C07227=1047.731,387.516,-124.764,173.908,41.828,158.146
C07228=1047.739,387.762,-124.805,173.915,41.833,158.148
C07229=1047.748,388.008,-124.847,173.922,41.839,158.150
C07230=1047.757,388.255,-124.889,173.929,41.845,158.152
C07231=1047.766,388.500,-124.931,173.936,41.851,158.154
C07232=1047.773,388.746,-124.973,173.943,41.857,158.155
C07233=1047.782,388.993,-125.015,173.951,41.863,158.157
C07234=1047.791,389.239,-125.057,173.957,41.869,158.159
C07235=1047.799,389.482,-125.099,173.964,41.874,158.161
C07236=1047.807,389.726,-125.140,173.972,41.880,158.163
C07237=1047.816,389.969,-125.182,173.979,41.887,158.165
C07238=1047.824,390.213,-125.224,173.985,41.893,158.167
C07239=1047.833,390.456,-125.266,173.992,41.898,158.169
C07240=1047.840,390.700,-125.307,174.000,41.904,158.171
C07241=1047.849,390.943,-125.350,174.007,41.910,158.173
C07242=1047.858,391.187,-125.392,174.014,41.917,158.175
C07243=1047.871,391.561,-125.456,174.025,41.926,158.178
C07244=1047.884,391.936,-125.521,174.036,41.935,158.181
C07245=1047.896,392.311,-125.586,174.047,41.944,158.184
C07246=1047.910,392.686,-125.651,174.058,41.954,158.187
C07247=1047.918,392.932,-125.693,174.065,41.960,158.189
C07248=1047.927,393.178,-125.736,174.073,41.966,158.191
C07249=1047.936,393.424,-125.779,174.080,41.972,158.193
C07250=1047.944,393.670,-125.822,174.088,41.979,158.195
C07251=1047.953,393.916,-125.865,174.095,41.985,158.197
C07252=1047.961,394.163,-125.907,174.103,41.991,158.199
C07253=1047.970,394.409,-125.950,174.110,41.997,158.201
C07254=1047.979,394.655,-125.993,174.118,42.004,158.203
C07255=1047.987,394.901,-126.036,174.125,42.010,158.205
C07256=1047.996,395.147,-126.079,174.133,42.017,158.207
C07257=1048.004,395.393,-126.122,174.140,42.023,158.209
C07258=1048.013,395.639,-126.165,174.148,42.029,158.212
C07259=1048.022,395.885,-126.207,174.155,42.035,158.214
C07260=1048.031,396.131,-126.251,174.163,42.042,158.216
C07261=1048.040,396.377,-126.294,174.170,42.048,158.218
C07262=1048.048,396.623,-126.337,174.178,42.055,158.220
C07263=1048.057,396.869,-126.380,174.185,42.062,158.222
C07264=1048.066,397.114,-126.424,174.193,42.068,158.224
C07265=1048.074,397.360,-126.467,174.200,42.074,158.226
C07266=1048.083,397.607,-126.510,174.209,42.081,158.228
C07267=1048.092,397.853,-126.554,174.217,42.087,158.231
C07268=1048.101,398.099,-126.597,174.224,42.094,158.233
C07269=1048.109,398.344,-126.641,174.232,42.101,158.235
C07270=1048.119,398.591,-126.684,174.240,42.107,158.237
C07271=1048.127,398.836,-126.728,174.247,42.114,158.239
C07272=1048.136,399.082,-126.771,174.255,42.121,158.242
C07273=1048.145,399.328,-126.815,174.263,42.127,158.244
C07274=1048.154,399.574,-126.858,174.271,42.134,158.246
C07275=1048.162,399.821,-126.903,174.279,42.141,158.248
C07276=1048.171,400.066,-126.947,174.287,42.147,158.250
C07277=1048.180,400.312,-126.990,174.294,42.154,158.253
C07278=1048.189,400.559,-127.034,174.303,42.161,158.255
C07279=1048.198,400.804,-127.078,174.311,42.167,158.257
C07280=1048.207,401.050,-127.122,174.318,42.174,158.259
C07281=1048.216,401.296,-127.165,174.326,42.181,158.262
C07282=1048.225,401.542,-127.209,174.335,42.188,158.264
C07283=1048.234,401.788,-127.253,174.343,42.195,158.266
C07284=1048.243,402.034,-127.297,174.350,42.201,158.268
C07285=1048.252,402.280,-127.341,174.359,42.208,158.271
C07286=1048.261,402.526,-127.385,174.367,42.215,158.273
C07287=1048.270,402.772,-127.429,174.375,42.222,158.275
C07288=1048.279,403.018,-127.474,174.384,42.229,158.278
C07289=1048.288,403.264,-127.518,174.391,42.236,158.280
C07290=1048.298,403.509,-127.563,174.399,42.243,158.282
C07291=1048.311,403.897,-127.633,174.413,42.254,158.286
C07292=1048.326,404.285,-127.702,174.425,42.265,158.290
C07293=1048.340,404.673,-127.773,174.439,42.276,158.294
C07294=1048.354,405.061,-127.843,174.452,42.288,158.297
C07295=1048.363,405.308,-127.887,174.461,42.295,158.300
C07296=1048.372,405.553,-127.932,174.468,42.302,158.302
C07297=1048.381,405.799,-127.978,174.478,42.309,158.305
C07298=1048.390,406.044,-128.021,174.485,42.316,158.307
C07299=1048.399,406.290,-128.067,174.495,42.324,158.310
C07300=1048.409,406.536,-128.111,174.502,42.331,158.312
C07301=1048.417,406.782,-128.156,174.511,42.338,158.314
C07302=1048.427,407.028,-128.201,174.519,42.345,158.317
C07303=1048.436,407.274,-128.246,174.528,42.353,158.319
C07304=1048.446,407.520,-128.291,174.537,42.360,158.322
C07305=1048.455,407.765,-128.336,174.545,42.367,158.324
C07306=1048.464,408.011,-128.381,174.555,42.374,158.327
C07307=1048.473,408.257,-128.426,174.563,42.382,158.329
C07308=1048.483,408.502,-128.471,174.572,42.389,158.332
C07309=1048.492,408.748,-128.517,174.580,42.397,158.334
C07310=1048.502,408.994,-128.561,174.589,42.404,158.337
C07311=1048.511,409.239,-128.607,174.598,42.412,158.339
C07312=1048.520,409.485,-128.652,174.606,42.419,158.342
C07313=1048.529,409.731,-128.697,174.615,42.427,158.344
C07314=1048.539,409.976,-128.742,174.625,42.434,158.347
C07315=1048.548,410.222,-128.787,174.633,42.442,158.350
C07316=1048.557,410.468,-128.833,174.642,42.449,158.352
C07317=1048.567,410.714,-128.878,174.651,42.456,158.355
C07318=1048.577,410.959,-128.924,174.660,42.464,158.357
C07319=1048.586,411.205,-128.969,174.669,42.472,158.360
C07320=1048.595,411.451,-129.014,174.678,42.479,158.362
C07321=1048.606,411.696,-129.060,174.687,42.487,158.365
C07322=1048.615,411.942,-129.106,174.696,42.495,158.368
C07323=1048.624,412.187,-129.152,174.705,42.502,158.370
C07324=1048.635,412.433,-129.197,174.715,42.510,158.373
C07325=1048.643,412.679,-129.242,174.724,42.518,158.376
C07326=1048.653,412.925,-129.288,174.732,42.526,158.378
C07327=1048.663,413.170,-129.335,174.742,42.534,158.381
C07328=1048.672,413.416,-129.380,174.751,42.541,158.384
C07329=1048.682,413.662,-129.426,174.761,42.549,158.387
C07330=1048.692,413.907,-129.472,174.770,42.557,158.389
C07331=1048.701,414.152,-129.519,174.779,42.565,158.392
C07332=1048.711,414.398,-129.565,174.789,42.573,158.395
C07333=1048.720,414.643,-129.611,174.798,42.581,158.397
C07334=1048.730,414.889,-129.658,174.807,42.589,158.400
C07335=1048.739,415.134,-129.704,174.817,42.597,158.403
C07336=1048.749,415.380,-129.750,174.826,42.604,158.406
C07337=1048.758,415.626,-129.796,174.836,42.613,158.409
C07338=1048.769,415.871,-129.842,174.845,42.621,158.411
C07339=1048.778,416.116,-129.889,174.855,42.629,158.414
C07340=1048.788,416.362,-129.935,174.864,42.637,158.417
C07341=1048.797,416.607,-129.981,174.874,42.645,158.420
C07342=1048.808,416.853,-130.028,174.883,42.653,158.423
C07343=1048.817,417.099,-130.075,174.893,42.662,158.425
C07344=1048.827,417.344,-130.121,174.903,42.669,158.428
C07345=1048.837,417.589,-130.168,174.913,42.678,158.431
C07346=1048.847,417.835,-130.215,174.923,42.686,158.434
C07347=1048.862,418.230,-130.290,174.939,42.699,158.439
C07348=1048.879,418.625,-130.365,174.954,42.712,158.443
C07349=1048.895,419.020,-130.441,174.970,42.726,158.448
C07350=1048.911,419.415,-130.517,174.986,42.740,158.453
C07351=1048.921,419.660,-130.563,174.996,42.748,158.456
C07352=1048.930,419.906,-130.611,175.007,42.756,158.459
C07353=1048.940,420.152,-130.658,175.017,42.765,158.462
C07354=1048.950,420.397,-130.705,175.026,42.774,158.465
C07355=1048.960,420.642,-130.752,175.037,42.782,158.468
C07356=1048.971,420.887,-130.799,175.047,42.791,158.471
C07357=1048.980,421.133,-130.847,175.058,42.799,158.474
C07358=1048.990,421.378,-130.894,175.068,42.808,158.477
C07359=1049.001,421.623,-130.942,175.078,42.816,158.480
C07360=1049.011,421.868,-130.990,175.088,42.825,158.483
C07361=1049.020,422.114,-131.037,175.098,42.834,158.486
C07362=1049.031,422.359,-131.085,175.109,42.842,158.489
C07363=1049.041,422.604,-131.132,175.119,42.851,158.492
C07364=1049.051,422.849,-131.180,175.130,42.860,158.495
C07365=1049.061,423.094,-131.227,175.141,42.868,158.499
C07366=1049.071,423.339,-131.275,175.151,42.878,158.502
C07367=1049.082,423.585,-131.323,175.162,42.886,158.505
C07368=1049.093,423.830,-131.371,175.172,42.895,158.508
C07369=1049.103,424.075,-131.418,175.183,42.904,158.511
C07370=1049.112,424.320,-131.467,175.194,42.913,158.514
C07371=1049.123,424.566,-131.514,175.204,42.922,158.518
C07372=1049.134,424.811,-131.562,175.215,42.931,158.521
C07373=1049.144,425.056,-131.611,175.226,42.939,158.524
C07374=1049.154,425.302,-131.658,175.236,42.949,158.527
C07375=1049.165,425.546,-131.706,175.247,42.957,158.530
C07376=1049.175,425.792,-131.755,175.259,42.966,158.534
C07377=1049.186,426.037,-131.803,175.270,42.976,158.537
C07378=1049.195,426.282,-131.852,175.280,42.985,158.540
C07379=1049.207,426.527,-131.900,175.291,42.994,158.544
C07380=1049.216,426.772,-131.948,175.303,43.003,158.547
C07381=1049.227,427.017,-131.997,175.314,43.012,158.550
C07382=1049.237,427.262,-132.046,175.325,43.021,158.554
C07383=1049.249,427.507,-132.094,175.336,43.031,158.557
C07384=1049.258,427.752,-132.143,175.348,43.040,158.560
C07385=1049.269,427.997,-132.191,175.359,43.049,158.564
C07386=1049.279,428.242,-132.240,175.369,43.059,158.567
C07387=1049.291,428.487,-132.289,175.381,43.068,158.571
C07388=1049.301,428.732,-132.338,175.392,43.078,158.574
C07389=1049.311,428.977,-132.387,175.403,43.087,158.577
C07390=1049.322,429.222,-132.436,175.416,43.096,158.581
C07391=1049.332,429.467,-132.484,175.427,43.106,158.584
C07392=1049.344,429.712,-132.533,175.439,43.116,158.588
C07393=1049.354,429.957,-132.583,175.450,43.125,158.591
C07394=1049.365,430.202,-132.633,175.462,43.135,158.595
C07395=1049.375,430.447,-132.681,175.473,43.144,158.599
C07396=1049.385,430.692,-132.731,175.485,43.154,158.602
C07397=1049.397,430.937,-132.780,175.496,43.163,158.606
C07398=1049.407,431.182,-132.829,175.508,43.173,158.609
C07399=1049.417,431.426,-132.879,175.521,43.183,158.613
C07400=1049.428,431.671,-132.928,175.532,43.193,158.616
C07401=1049.440,431.915,-132.978,175.544,43.203,158.620
C07402=1049.451,432.160,-133.027,175.557,43.212,158.624
C07403=1049.459,432.370,-133.070,175.567,43.221,158.627
C07404=1049.469,432.579,-133.112,175.577,43.229,158.630
C07405=1049.478,432.788,-133.155,175.587,43.237,158.633
C07406=1049.487,432.997,-133.197,175.598,43.246,158.636
C07407=1049.498,433.207,-133.240,175.608,43.254,158.639
C07408=1049.507,433.416,-133.283,175.618,43.263,158.642
C07409=1049.516,433.625,-133.325,175.629,43.271,158.646
C07410=1049.525,433.834,-133.368,175.639,43.280,158.649
C07411=1049.536,434.079,-133.417,175.651,43.290,158.653
C07412=1049.547,434.323,-133.467,175.664,43.300,158.656
C07413=1049.559,434.569,-133.518,175.676,43.310,158.660
C07414=1049.570,434.813,-133.568,175.689,43.320,158.664
C07415=1049.581,435.058,-133.618,175.702,43.330,158.668
C07416=1049.592,435.302,-133.668,175.714,43.341,158.672
C07417=1049.604,435.547,-133.718,175.726,43.351,158.675
C07418=1049.615,435.792,-133.769,175.739,43.361,158.679
C07419=1049.626,436.036,-133.819,175.752,43.371,158.683
C07420=1049.637,436.281,-133.870,175.764,43.381,158.687
C07421=1049.648,436.526,-133.920,175.778,43.391,158.691
C07422=1049.659,436.770,-133.970,175.790,43.402,158.695
C07423=1049.671,437.015,-134.021,175.803,43.412,158.699
C07424=1049.682,437.259,-134.072,175.816,43.423,158.703
C07425=1049.694,437.504,-134.123,175.829,43.433,158.707
C07426=1049.705,437.749,-134.173,175.841,43.444,158.711
C07427=1049.717,437.993,-134.224,175.855,43.455,158.715
C07428=1049.728,438.238,-134.275,175.868,43.465,158.719
C07429=1049.740,438.482,-134.326,175.881,43.476,158.723
C07430=1049.750,438.727,-134.376,175.894,43.486,158.727
C07431=1049.762,438.971,-134.428,175.908,43.497,158.731
C07432=1049.774,439.216,-134.480,175.921,43.508,158.735
C07433=1049.785,439.460,-134.531,175.935,43.518,158.739
C07434=1049.797,439.704,-134.582,175.948,43.529,158.743
C07435=1049.808,439.949,-134.633,175.961,43.540,158.747
C07436=1049.820,440.193,-134.684,175.975,43.551,158.751
C07437=1049.831,440.438,-134.736,175.988,43.562,158.756
C07438=1049.843,440.682,-134.788,176.002,43.573,158.760
C07439=1049.855,440.926,-134.840,176.016,43.583,158.764
C07440=1049.866,441.170,-134.891,176.030,43.594,158.768
C07441=1049.878,441.415,-134.942,176.043,43.605,158.772
C07442=1049.890,441.659,-134.993,176.057,43.616,158.777
C07443=1049.901,441.903,-135.046,176.072,43.627,158.781
C07444=1049.913,442.148,-135.098,176.085,43.639,158.785
C07445=1049.925,442.392,-135.150,176.099,43.650,158.790
C07446=1049.936,442.637,-135.202,176.114,43.661,158.794
C07447=1049.949,442.880,-135.254,176.128,43.672,158.798
C07448=1049.961,443.124,-135.306,176.141,43.683,158.803
C07449=1049.973,443.369,-135.357,176.156,43.695,158.807
C07450=1049.984,443.613,-135.410,176.170,43.706,158.812
C07451=1049.996,443.857,-135.462,176.185,43.717,158.816
C07452=1050.009,444.101,-135.514,176.199,43.729,158.821
C07453=1050.020,444.345,-135.567,176.214,43.740,158.825
C07454=1050.033,444.590,-135.619,176.229,43.752,158.830
C07455=1050.045,444.834,-135.672,176.243,43.763,158.834
C07456=1050.056,445.078,-135.724,176.258,43.775,158.839
C07457=1050.069,445.322,-135.777,176.273,43.786,158.843
C07458=1050.081,445.566,-135.829,176.287,43.798,158.848
C07459=1050.093,445.809,-135.881,176.302,43.809,158.852
C07460=1050.106,446.052,-135.934,176.317,43.821,158.857
C07461=1050.119,446.296,-135.986,176.332,43.832,158.862
C07462=1050.132,446.540,-136.038,176.347,43.843,158.866
C07463=1050.148,446.805,-136.093,176.364,43.856,158.871
C07464=1050.165,447.073,-136.149,176.380,43.868,158.876
C07465=1050.182,447.340,-136.203,176.396,43.879,158.881
C07466=1050.201,447.608,-136.257,176.414,43.891,158.886
C07467=1050.219,447.852,-136.306,176.430,43.901,158.890
C07468=1050.237,448.096,-136.353,176.444,43.912,158.894
C07469=1050.255,448.341,-136.401,176.460,43.922,158.899
C07470=1050.275,448.586,-136.448,176.476,43.932,158.903
C07471=1050.296,448.830,-136.495,176.492,43.942,158.907
C07472=1050.317,449.075,-136.541,176.508,43.951,158.911
C07473=1050.338,449.321,-136.586,176.523,43.961,158.916
C07474=1050.361,449.566,-136.631,176.540,43.971,158.920
C07475=1050.384,449.811,-136.675,176.556,43.980,158.924
C07476=1050.408,450.056,-136.719,176.572,43.989,158.928
C07477=1050.432,450.302,-136.762,176.588,43.998,158.932
C07478=1050.458,450.546,-136.805,176.605,44.007,158.936
C07479=1050.144,450.574,-137.105,176.604,44.099,158.963
C07480=1050.118,450.329,-137.062,176.588,44.090,158.959
C07481=1050.094,450.083,-137.019,176.572,44.081,158.955
C07482=1050.070,449.838,-136.975,176.556,44.073,158.951
C07483=1050.046,449.593,-136.931,176.539,44.064,158.947
C07484=1050.024,449.348,-136.887,176.523,44.054,158.942
C07485=1050.002,449.103,-136.841,176.507,44.044,158.938
C07486=1049.981,448.858,-136.795,176.492,44.034,158.934
C07487=1049.960,448.613,-136.749,176.475,44.025,158.930
C07488=1049.941,448.368,-136.702,176.460,44.015,158.925
C07489=1049.921,448.124,-136.654,176.444,44.005,158.921
C07490=1049.903,447.880,-136.607,176.428,43.995,158.917
C07491=1049.886,447.636,-136.558,176.412,43.985,158.912
C07492=1049.868,447.386,-136.507,176.397,43.973,158.908
C07493=1049.851,447.137,-136.457,176.381,43.963,158.903
C07494=1049.836,446.888,-136.406,176.365,43.952,158.899
C07495=1049.821,446.639,-136.354,176.350,43.940,158.894
C07496=1049.806,446.395,-136.303,176.335,43.929,158.890
C07497=1049.792,446.151,-136.251,176.320,43.918,158.885
C07498=1049.779,445.908,-136.199,176.305,43.907,158.881
C07499=1049.767,445.666,-136.147,176.290,43.895,158.876
C07500=1049.755,445.422,-136.094,176.275,43.884,158.871
C07501=1049.743,445.177,-136.041,176.260,43.872,158.867
C07502=1049.730,444.933,-135.989,176.246,43.861,158.862
C07503=1049.719,444.690,-135.936,176.231,43.850,158.858
C07504=1049.706,444.446,-135.884,176.216,43.838,158.853
C07505=1049.694,444.201,-135.831,176.202,43.826,158.849
C07506=1049.682,443.957,-135.779,176.187,43.816,158.844
C07507=1049.670,443.713,-135.726,176.173,43.804,158.840
C07508=1049.658,443.469,-135.675,176.158,43.793,158.835
C07509=1049.647,443.224,-135.622,176.144,43.782,158.831
C07510=1049.635,442.980,-135.570,176.129,43.770,158.826
C07511=1049.622,442.737,-135.518,176.115,43.759,158.822
C07512=1049.611,442.492,-135.466,176.101,43.748,158.818
C07513=1049.599,442.248,-135.414,176.087,43.737,158.813
C07514=1049.587,442.003,-135.363,176.072,43.726,158.809
C07515=1049.575,441.759,-135.310,176.059,43.715,158.805
C07516=1049.564,441.515,-135.258,176.045,43.704,158.800
C07517=1049.552,441.270,-135.207,176.030,43.693,158.796
C07518=1049.540,441.026,-135.155,176.017,43.682,158.792
C07519=1049.528,440.782,-135.104,176.003,43.672,158.788
C07520=1049.516,440.537,-135.052,175.989,43.660,158.783
C07521=1049.504,440.293,-135.001,175.976,43.650,158.779
C07522=1049.494,440.049,-134.949,175.962,43.639,158.775
C07523=1049.482,439.804,-134.898,175.948,43.628,158.771
C07524=1049.470,439.560,-134.846,175.935,43.618,158.767
C07525=1049.458,439.316,-134.795,175.921,43.607,158.763
C07526=1049.447,439.071,-134.744,175.908,43.596,158.759
C07527=1049.435,438.826,-134.693,175.894,43.585,158.754
C07528=1049.424,438.582,-134.642,175.881,43.575,158.750
C07529=1049.413,438.337,-134.590,175.868,43.564,158.746
C07530=1049.401,438.092,-134.539,175.855,43.554,158.742
C07531=1049.390,437.849,-134.488,175.841,43.543,158.738
C07532=1049.378,437.603,-134.438,175.829,43.533,158.734
C07533=1049.367,437.360,-134.387,175.816,43.522,158.730
C07534=1049.355,437.114,-134.336,175.803,43.512,158.726
C07535=1049.344,436.870,-134.286,175.789,43.502,158.722
C07536=1049.333,436.626,-134.235,175.776,43.492,158.718
C07537=1049.322,436.381,-134.184,175.764,43.481,158.715
C07538=1049.311,436.137,-134.134,175.751,43.471,158.711
C07539=1049.299,435.892,-134.083,175.738,43.460,158.707
C07540=1049.287,435.647,-134.033,175.725,43.451,158.703
C07541=1049.276,435.403,-133.983,175.713,43.440,158.699
C07542=1049.265,435.158,-133.932,175.700,43.430,158.695
C07543=1049.254,434.913,-133.883,175.687,43.420,158.691
C07544=1049.243,434.668,-133.832,175.675,43.410,158.688
C07545=1049.231,434.424,-133.782,175.662,43.400,158.684
C07546=1049.220,434.180,-133.732,175.650,43.390,158.680
C07547=1049.209,433.934,-133.682,175.637,43.380,158.676
C07548=1049.200,433.724,-133.639,175.627,43.372,158.673
C07549=1049.190,433.514,-133.596,175.616,43.363,158.670
C07550=1049.180,433.304,-133.554,175.606,43.355,158.667
C07551=1049.171,433.094,-133.511,175.596,43.346,158.663
C07552=1049.161,432.884,-133.468,175.585,43.338,158.660
C07553=1049.152,432.673,-133.425,175.574,43.329,158.657
C07554=1049.143,432.463,-133.382,175.563,43.321,158.654
C07555=1049.134,432.253,-133.340,175.553,43.313,158.651
C07556=1049.123,432.008,-133.290,175.542,43.302,158.647
C07557=1049.112,431.764,-133.241,175.530,43.293,158.644
C07558=1049.101,431.519,-133.191,175.517,43.283,158.640
C07559=1049.090,431.274,-133.141,175.506,43.273,158.636
C07560=1049.080,431.029,-133.092,175.494,43.264,158.633
C07561=1049.068,430.784,-133.043,175.482,43.254,158.629
C07562=1049.058,430.539,-132.993,175.470,43.244,158.626
C07563=1049.048,430.294,-132.944,175.458,43.235,158.622
C07564=1049.037,430.049,-132.894,175.447,43.225,158.618
C07565=1049.026,429.804,-132.846,175.435,43.216,158.615
C07566=1049.015,429.559,-132.796,175.424,43.207,158.612
C07567=1049.005,429.315,-132.747,175.412,43.197,158.608
C07568=1048.994,429.070,-132.698,175.401,43.187,158.605
C07569=1048.983,428.824,-132.649,175.389,43.178,158.601
C07570=1048.973,428.578,-132.600,175.377,43.169,158.598
C07571=1048.962,428.334,-132.552,175.366,43.160,158.594
C07572=1048.952,428.089,-132.503,175.354,43.150,158.591
C07573=1048.941,427.845,-132.454,175.343,43.141,158.587
C07574=1048.931,427.599,-132.405,175.332,43.132,158.584
C07575=1048.920,427.354,-132.357,175.321,43.123,158.581
C07576=1048.909,427.109,-132.308,175.310,43.113,158.577
C07577=1048.898,426.864,-132.259,175.298,43.104,158.574
C07578=1048.889,426.619,-132.211,175.287,43.095,158.571
C07579=1048.878,426.374,-132.163,175.276,43.086,158.567
C07580=1048.868,426.129,-132.114,175.265,43.077,158.564
C07581=1048.857,425.884,-132.066,175.254,43.068,158.561
C07582=1048.847,425.638,-132.017,175.243,43.059,158.557
C07583=1048.836,425.394,-131.969,175.232,43.050,158.554
C07584=1048.826,425.149,-131.921,175.221,43.041,158.551
C07585=1048.816,424.903,-131.872,175.210,43.032,158.548
C07586=1048.805,424.658,-131.825,175.200,43.023,158.545
C07587=1048.794,424.413,-131.777,175.189,43.014,158.541
C07588=1048.785,424.168,-131.728,175.178,43.005,158.538
C07589=1048.774,423.922,-131.681,175.168,42.997,158.535
C07590=1048.764,423.678,-131.633,175.157,42.988,158.532
C07591=1048.753,423.432,-131.586,175.146,42.979,158.529
C07592=1048.743,423.187,-131.537,175.135,42.970,158.525
C07593=1048.733,422.942,-131.490,175.124,42.961,158.522
C07594=1048.723,422.697,-131.442,175.114,42.953,158.519
C07595=1048.712,422.452,-131.395,175.104,42.944,158.516
C07596=1048.703,422.206,-131.347,175.093,42.936,158.513
C07597=1048.693,421.961,-131.300,175.083,42.927,158.510
C07598=1048.682,421.716,-131.252,175.072,42.918,158.507
C07599=1048.671,421.470,-131.204,175.062,42.910,158.504
C07600=1048.661,421.225,-131.157,175.052,42.901,158.501
C07601=1048.652,420.980,-131.110,175.041,42.893,158.498
C07602=1048.642,420.735,-131.062,175.031,42.884,158.495
C07603=1048.632,420.489,-131.015,175.020,42.876,158.491
C07604=1048.622,420.244,-130.968,175.011,42.867,158.489
C07605=1048.612,419.999,-130.921,175.001,42.859,158.486
C07606=1048.602,419.753,-130.873,174.990,42.850,158.482
C07607=1048.592,419.508,-130.826,174.980,42.842,158.480
C07608=1048.576,419.111,-130.750,174.964,42.828,158.475
C07609=1048.560,418.714,-130.674,174.947,42.815,158.470
C07610=1048.544,418.317,-130.598,174.931,42.801,158.465
C07611=1048.528,417.920,-130.523,174.915,42.788,158.461
C07612=1048.517,417.674,-130.476,174.906,42.780,158.458
C07613=1048.508,417.429,-130.429,174.896,42.772,158.455
C07614=1048.498,417.183,-130.383,174.886,42.764,158.452
C07615=1048.488,416.938,-130.336,174.876,42.756,158.449
C07616=1048.478,416.692,-130.289,174.866,42.748,158.446
C07617=1048.468,416.446,-130.243,174.857,42.740,158.443
C07618=1048.459,416.202,-130.196,174.847,42.731,158.441
C07619=1048.449,415.956,-130.149,174.838,42.724,158.438
C07620=1048.440,415.711,-130.103,174.828,42.715,158.435
C07621=1048.430,415.465,-130.057,174.819,42.707,158.432
C07622=1048.419,415.219,-130.011,174.809,42.700,158.429
C07623=1048.410,414.974,-129.965,174.800,42.692,158.427
C07624=1048.400,414.728,-129.918,174.790,42.684,158.424
C07625=1048.391,414.483,-129.872,174.781,42.676,158.421
C07626=1048.381,414.238,-129.826,174.771,42.668,158.418
C07627=1048.371,413.992,-129.779,174.762,42.660,158.416
C07628=1048.362,413.746,-129.733,174.753,42.652,158.413
C07629=1048.352,413.501,-129.687,174.743,42.645,158.410
C07630=1048.343,413.255,-129.641,174.734,42.637,158.407
C07631=1048.333,413.010,-129.596,174.724,42.629,158.405
C07632=1048.323,412.764,-129.549,174.715,42.621,158.402
C07633=1048.314,412.518,-129.504,174.706,42.614,158.399
C07634=1048.304,412.272,-129.457,174.696,42.606,158.397
C07635=1048.295,412.027,-129.413,174.687,42.598,158.394
C07636=1048.285,411.781,-129.366,174.679,42.590,158.391
C07637=1048.275,411.535,-129.321,174.670,42.583,158.389
C07638=1048.266,411.289,-129.276,174.660,42.575,158.386
C07639=1048.257,411.044,-129.230,174.651,42.568,158.384
C07640=1048.247,410.799,-129.185,174.642,42.560,158.381
C07641=1048.238,410.552,-129.139,174.634,42.553,158.378
C07642=1048.228,410.307,-129.094,174.625,42.545,158.376
C07643=1048.219,410.061,-129.048,174.615,42.538,158.373
C07644=1048.209,409.816,-129.003,174.606,42.530,158.371
C07645=1048.200,409.570,-128.958,174.598,42.523,158.368
C07646=1048.190,409.325,-128.913,174.589,42.515,158.365
C07647=1048.181,409.078,-128.867,174.580,42.508,158.363
C07648=1048.171,408.833,-128.822,174.570,42.500,158.360
C07649=1048.162,408.587,-128.777,174.562,42.493,158.358
C07650=1048.152,408.341,-128.732,174.553,42.486,158.355
C07651=1048.143,408.095,-128.687,174.545,42.479,158.353
C07652=1048.134,407.850,-128.641,174.536,42.471,158.350
C07653=1048.125,407.604,-128.597,174.527,42.464,158.348
C07654=1048.116,407.358,-128.551,174.519,42.457,158.345
C07655=1048.106,407.112,-128.507,174.510,42.449,158.343
C07656=1048.097,406.866,-128.462,174.502,42.442,158.341
C07657=1048.088,406.622,-128.417,174.493,42.435,158.338
C07658=1048.079,406.376,-128.372,174.484,42.428,158.336
C07659=1048.070,406.130,-128.328,174.476,42.420,158.333
C07660=1048.061,405.884,-128.282,174.467,42.414,158.331
C07661=1048.051,405.638,-128.238,174.459,42.407,158.328
C07662=1048.042,405.392,-128.193,174.450,42.399,158.326
C07663=1048.034,405.146,-128.149,174.442,42.392,158.323
C07664=1048.019,404.757,-128.078,174.428,42.381,158.320
C07665=1048.004,404.366,-128.007,174.415,42.370,158.316
C07666=1047.990,403.976,-127.936,174.402,42.359,158.312
C07667=1047.976,403.586,-127.866,174.389,42.348,158.308
C07668=1047.967,403.341,-127.822,174.380,42.341,158.306
C07669=1047.958,403.095,-127.777,174.373,42.334,158.304
C07670=1047.948,402.849,-127.733,174.364,42.327,158.301
C07671=1047.940,402.603,-127.689,174.356,42.320,158.299
C07672=1047.931,402.357,-127.645,174.348,42.313,158.297
C07673=1047.921,402.111,-127.600,174.339,42.306,158.295
C07674=1047.913,401.865,-127.557,174.331,42.299,158.292
C07675=1047.903,401.619,-127.513,174.324,42.293,158.290
C07676=1047.894,401.374,-127.469,174.315,42.286,158.288
C07677=1047.886,401.127,-127.424,174.307,42.279,158.285
C07678=1047.877,400.882,-127.380,174.299,42.272,158.283
C07679=1047.868,400.635,-127.337,174.292,42.266,158.281
C07680=1047.859,400.389,-127.293,174.283,42.259,158.279
C07681=1047.850,400.143,-127.249,174.275,42.252,158.276
C07682=1047.841,399.898,-127.205,174.267,42.246,158.274
C07683=1047.832,399.651,-127.162,174.260,42.239,158.272
C07684=1047.823,399.406,-127.118,174.251,42.232,158.270
C07685=1047.814,399.160,-127.075,174.243,42.226,158.268
C07686=1047.805,398.914,-127.031,174.236,42.219,158.265
C07687=1047.796,398.668,-126.987,174.228,42.213,158.263
C07688=1047.788,398.422,-126.944,174.220,42.206,158.261
C07689=1047.778,398.176,-126.900,174.213,42.199,158.259
C07690=1047.770,397.930,-126.857,174.204,42.193,158.257
C07691=1047.761,397.684,-126.814,174.197,42.187,158.254
C07692=1047.752,397.438,-126.770,174.189,42.180,158.252
C07693=1047.743,397.192,-126.727,174.181,42.173,158.250
C07694=1047.735,396.946,-126.683,174.174,42.167,158.248
C07695=1047.726,396.700,-126.640,174.166,42.160,158.246
C07696=1047.718,396.454,-126.597,174.159,42.154,158.244
C07697=1047.708,396.207,-126.554,174.151,42.148,158.242
C07698=1047.700,395.962,-126.510,174.143,42.141,158.239
C07699=1047.691,395.716,-126.467,174.135,42.135,158.237
C07700=1047.683,395.470,-126.424,174.127,42.129,158.235
C07701=1047.673,395.224,-126.382,174.120,42.122,158.233
C07702=1047.665,394.978,-126.339,174.112,42.116,158.231
C07703=1047.656,394.732,-126.296,174.105,42.110,158.229
C07704=1047.647,394.485,-126.252,174.097,42.104,158.227
C07705=1047.639,394.239,-126.209,174.090,42.097,158.225
C07706=1047.630,393.993,-126.167,174.082,42.091,158.223
C07707=1047.621,393.747,-126.124,174.075,42.085,158.221
C07708=1047.613,393.501,-126.081,174.067,42.078,158.219
C07709=1047.604,393.255,-126.038,174.060,42.072,158.217
C07710=1047.596,393.009,-125.995,174.052,42.066,158.215
C07711=1047.587,392.763,-125.953,174.045,42.060,158.213
C07712=1047.578,392.517,-125.910,174.039,42.054,158.211
C07713=1047.571,392.271,-125.868,174.031,42.047,158.209
C07714=1047.562,392.025,-125.825,174.024,42.041,158.207
C07715=1047.553,391.779,-125.782,174.016,42.035,158.205
C07716=1047.545,391.532,-125.740,174.009,42.029,158.203
C07717=1047.536,391.286,-125.697,174.001,42.023,158.201
C07718=1047.527,391.040,-125.655,173.994,42.017,158.199
C07719=1047.519,390.794,-125.612,173.987,42.011,158.197
C07720=1047.506,390.422,-125.549,173.976,42.002,158.194
C07721=1047.493,390.051,-125.485,173.966,41.993,158.191
C07722=1047.480,389.680,-125.422,173.954,41.984,158.188
C07723=1047.468,389.309,-125.358,173.944,41.975,158.185
C07724=1047.459,389.062,-125.316,173.936,41.970,158.183
C07725=1047.451,388.816,-125.273,173.930,41.963,158.181
C07726=1047.441,388.570,-125.231,173.923,41.957,158.179
C07727=1047.434,388.324,-125.189,173.916,41.952,158.177
C07728=1047.425,388.078,-125.147,173.908,41.946,158.175
C07729=1047.416,387.831,-125.106,173.901,41.940,158.174
C07730=1047.408,387.584,-125.063,173.895,41.935,158.172
C07731=1047.399,387.339,-125.022,173.888,41.928,158.170
C07732=1047.391,387.092,-124.980,173.880,41.923,158.168
C07733=1047.382,386.846,-124.938,173.873,41.917,158.166
C07734=1047.374,386.600,-124.897,173.867,41.911,158.164
C07735=1047.365,386.354,-124.855,173.860,41.906,158.162
C07736=1047.357,386.106,-124.813,173.853,41.900,158.160
C07737=1047.349,385.861,-124.772,173.845,41.894,158.159
C07738=1047.340,385.614,-124.730,173.839,41.888,158.157
C07739=1047.332,385.368,-124.688,173.832,41.883,158.155
C07740=1047.323,385.122,-124.647,173.825,41.877,158.153
C07741=1047.315,384.876,-124.606,173.819,41.872,158.151
C07742=1047.307,384.629,-124.564,173.811,41.866,158.149
C07743=1047.298,384.383,-124.522,173.805,41.860,158.148
C07744=1047.290,384.136,-124.481,173.798,41.855,158.146
C07745=1047.282,383.890,-124.439,173.791,41.849,158.144
C07746=1047.274,383.644,-124.398,173.785,41.844,158.142
C07747=1047.266,383.398,-124.357,173.778,41.838,158.140
C07748=1047.257,383.151,-124.315,173.771,41.832,158.139
C07749=1047.249,382.905,-124.274,173.764,41.827,158.137
C07750=1047.240,382.659,-124.232,173.757,41.821,158.135
C07751=1047.232,382.412,-124.192,173.751,41.816,158.133
C07752=1047.225,382.165,-124.150,173.744,41.810,158.132
C07753=1047.216,381.919,-124.109,173.738,41.805,158.130
C07754=1047.208,381.673,-124.068,173.731,41.799,158.128
C07755=1047.200,381.426,-124.026,173.725,41.794,158.126
C07756=1047.192,381.180,-123.985,173.718,41.789,158.125
C07757=1047.184,380.934,-123.945,173.712,41.783,158.123
C07758=1047.175,380.687,-123.904,173.705,41.778,158.121
C07759=1047.168,380.441,-123.862,173.699,41.772,158.119
C07760=1047.160,380.195,-123.821,173.692,41.766,158.118
C07761=1047.152,379.948,-123.780,173.686,41.761,158.116
C07762=1047.144,379.701,-123.739,173.679,41.756,158.114
C07763=1047.136,379.455,-123.698,173.673,41.751,158.112
C07764=1047.128,379.208,-123.657,173.666,41.745,158.111
C07765=1047.120,378.962,-123.617,173.660,41.740,158.109
C07766=1047.111,378.715,-123.576,173.653,41.735,158.107
C07767=1047.103,378.469,-123.535,173.647,41.730,158.106
C07768=1047.094,378.212,-123.492,173.640,41.724,158.104
C07769=1047.086,377.954,-123.450,173.634,41.718,158.102
C07770=1047.077,377.698,-123.408,173.626,41.713,158.100
C07771=1047.069,377.440,-123.366,173.620,41.708,158.099
C07772=1047.061,377.194,-123.325,173.614,41.703,158.097
C07773=1047.053,376.947,-123.285,173.608,41.697,158.096
C07774=1047.044,376.700,-123.244,173.601,41.692,158.094
C07775=1047.036,376.453,-123.204,173.595,41.687,158.092
C07776=1047.025,376.126,-123.151,173.586,41.680,158.090
C07777=1047.015,375.798,-123.097,173.578,41.673,158.088
C07778=1047.004,375.472,-123.043,173.569,41.667,158.086
C07779=1046.994,375.144,-122.989,173.562,41.659,158.083
C07780=1046.986,374.897,-122.950,173.555,41.654,158.082
C07781=1046.978,374.651,-122.909,173.549,41.649,158.080
C07782=1046.970,374.404,-122.869,173.543,41.645,158.079
C07783=1046.962,374.158,-122.829,173.536,41.640,158.077
C07784=1046.954,373.911,-122.789,173.530,41.634,158.076
C07785=1046.946,373.665,-122.748,173.524,41.629,158.074
C07786=1046.938,373.418,-122.708,173.518,41.624,158.072
C07787=1046.931,373.171,-122.668,173.512,41.620,158.071
C07788=1046.923,372.925,-122.628,173.506,41.614,158.069
C07789=1046.915,372.678,-122.588,173.500,41.609,158.068
C07790=1046.906,372.431,-122.548,173.493,41.604,158.066
C07791=1046.899,372.186,-122.508,173.487,41.599,158.064
C07792=1046.891,371.939,-122.468,173.482,41.594,158.063
C07793=1046.884,371.692,-122.428,173.476,41.589,158.061
C07794=1046.876,371.445,-122.388,173.470,41.584,158.060
C07795=1046.868,371.198,-122.348,173.463,41.579,158.058
C07796=1046.860,370.951,-122.308,173.457,41.575,158.057
C07797=1046.852,370.705,-122.269,173.452,41.570,158.055
C07798=1046.844,370.458,-122.229,173.446,41.565,158.054
C07799=1046.836,370.211,-122.190,173.439,41.560,158.052
C07800=1046.829,369.965,-122.150,173.433,41.555,158.051
C07801=1046.821,369.718,-122.110,173.428,41.551,158.049
C07802=1046.812,369.471,-122.071,173.422,41.546,158.048
C07803=1046.805,369.224,-122.031,173.416,41.541,158.046
C07804=1046.796,368.978,-121.992,173.409,41.536,158.045
C07805=1046.789,368.732,-121.952,173.404,41.532,158.043
C07806=1046.781,368.485,-121.913,173.398,41.527,158.042
C07807=1046.773,368.237,-121.874,173.392,41.522,158.040
C07808=1046.765,367.991,-121.834,173.386,41.517,158.039
C07809=1046.758,367.745,-121.795,173.381,41.512,158.037
C07810=1046.750,367.498,-121.755,173.375,41.508,158.036
C07811=1046.742,367.251,-121.716,173.369,41.503,158.034
C07812=1046.734,367.004,-121.676,173.363,41.499,158.033
C07813=1046.726,366.758,-121.637,173.357,41.494,158.031
C07814=1046.719,366.510,-121.598,173.351,41.489,158.030
C07815=1046.710,366.264,-121.559,173.346,41.484,158.028
C07816=1046.704,366.017,-121.520,173.340,41.479,158.027
C07817=1046.695,365.770,-121.481,173.334,41.475,158.025
C07818=1046.688,365.524,-121.441,173.328,41.470,158.024
C07819=1046.680,365.277,-121.403,173.323,41.466,158.023
C07820=1046.672,365.030,-121.363,173.317,41.461,158.021
C07821=1046.665,364.783,-121.324,173.312,41.457,158.020
C07822=1046.657,364.536,-121.285,173.306,41.452,158.018
C07823=1046.650,364.290,-121.246,173.300,41.447,158.017
C07824=1046.642,364.042,-121.207,173.295,41.443,158.015
C07825=1046.635,363.796,-121.168,173.289,41.438,158.014
C07826=1046.627,363.549,-121.129,173.283,41.433,158.013
C07827=1046.620,363.302,-121.090,173.278,41.429,158.011
C07828=1046.611,363.056,-121.051,173.272,41.424,158.010
C07829=1046.605,362.809,-121.012,173.267,41.420,158.008
C07830=1046.596,362.562,-120.973,173.261,41.415,158.007
C07831=1046.589,362.315,-120.935,173.255,41.411,158.006
C07832=1046.578,361.996,-120.885,173.248,41.405,158.004
C07833=1046.568,361.677,-120.835,173.240,41.399,158.002
C07834=1046.559,361.358,-120.785,173.233,41.393,158.000
C07835=1046.549,361.040,-120.735,173.226,41.388,157.998
C07836=1046.541,360.792,-120.696,173.221,41.384,157.997
C07837=1046.534,360.546,-120.658,173.215,41.379,157.996
C07838=1046.526,360.299,-120.620,173.210,41.375,157.994
C07839=1046.518,360.052,-120.581,173.204,41.370,157.993
C07840=1046.511,359.805,-120.543,173.199,41.366,157.992
C07841=1046.504,359.557,-120.504,173.194,41.362,157.990
C07842=1046.496,359.311,-120.466,173.188,41.357,157.989
C07843=1046.488,359.064,-120.428,173.183,41.353,157.988
C07844=1046.480,358.817,-120.389,173.177,41.348,157.986
C07845=1046.473,358.570,-120.351,173.172,41.344,157.985
C07846=1046.466,358.324,-120.312,173.166,41.340,157.984
C07847=1046.458,358.076,-120.274,173.161,41.336,157.982
C07848=1046.451,357.829,-120.236,173.155,41.331,157.981
C07849=1046.443,357.583,-120.198,173.151,41.327,157.980
C07850=1046.435,357.335,-120.160,173.145,41.323,157.978
C07851=1046.428,357.088,-120.122,173.140,41.319,157.977
C07852=1046.420,356.842,-120.083,173.134,41.314,157.976
C07853=1046.413,356.595,-120.046,173.129,41.310,157.974
C07854=1046.405,356.348,-120.007,173.123,41.306,157.973
C07855=1046.397,356.100,-119.970,173.118,41.302,157.972
C07856=1046.390,355.854,-119.931,173.113,41.297,157.971
C07857=1046.383,355.607,-119.894,173.108,41.293,157.969
C07858=1046.374,355.360,-119.855,173.102,41.289,157.968
C07859=1046.367,355.112,-119.818,173.097,41.285,157.967
C07860=1046.360,354.866,-119.779,173.092,41.281,157.966
C07861=1046.352,354.619,-119.742,173.086,41.277,157.964
C07862=1046.345,354.372,-119.704,173.082,41.272,157.963
C07863=1046.337,354.124,-119.666,173.076,41.268,157.962
C07864=1046.330,353.877,-119.628,173.071,41.264,157.960
C07865=1046.322,353.631,-119.590,173.065,41.260,157.959
C07866=1046.315,353.384,-119.553,173.061,41.256,157.958
C07867=1046.308,353.137,-119.515,173.055,41.252,157.957
C07868=1046.300,352.889,-119.477,173.050,41.247,157.955
C07869=1046.293,352.643,-119.439,173.045,41.243,157.954
C07870=1046.286,352.396,-119.402,173.040,41.240,157.953
C07871=1046.278,352.148,-119.364,173.035,41.235,157.952
C07872=1046.271,351.901,-119.326,173.029,41.231,157.950
C07873=1046.263,351.654,-119.289,173.024,41.227,157.949
C07874=1046.256,351.406,-119.251,173.020,41.223,157.948
C07875=1046.249,351.160,-119.213,173.014,41.219,157.947
C07876=1046.241,350.913,-119.176,173.009,41.215,157.945
C07877=1046.233,350.666,-119.139,173.004,41.211,157.944
C07878=1046.226,350.419,-119.101,172.999,41.207,157.943
C07879=1046.219,350.172,-119.063,172.994,41.203,157.942
C07880=1046.212,349.925,-119.026,172.989,41.199,157.941
C07881=1046.204,349.677,-118.988,172.984,41.195,157.939
C07882=1046.197,349.430,-118.952,172.979,41.191,157.938
C07883=1046.189,349.183,-118.915,172.973,41.187,157.937
C07884=1046.182,348.936,-118.877,172.969,41.183,157.936
C07885=1046.174,348.689,-118.840,172.963,41.179,157.935
C07886=1046.167,348.442,-118.803,172.958,41.176,157.933
C07887=1046.160,348.195,-118.765,172.954,41.171,157.932
C07888=1046.151,347.882,-118.718,172.947,41.167,157.931
C07889=1046.141,347.569,-118.671,172.941,41.161,157.929
C07890=1046.132,347.255,-118.625,172.935,41.157,157.928
C07891=1046.123,346.941,-118.578,172.928,41.151,157.926
C07892=1046.116,346.694,-118.540,172.924,41.148,157.925
C07893=1046.108,346.447,-118.503,172.919,41.144,157.924
C07894=1046.101,346.200,-118.467,172.914,41.140,157.923
C07895=1046.094,345.953,-118.429,172.909,41.136,157.922
C07896=1046.086,345.706,-118.393,172.904,41.133,157.920
C07897=1046.079,345.459,-118.355,172.899,41.128,157.919
C07898=1046.071,345.212,-118.319,172.894,41.125,157.918
C07899=1046.064,344.964,-118.282,172.890,41.121,157.917
C07900=1046.057,344.718,-118.245,172.884,41.117,157.916
C07901=1046.050,344.470,-118.208,172.879,41.113,157.915
C07902=1046.043,344.223,-118.171,172.875,41.110,157.913
C07903=1046.035,343.975,-118.135,172.870,41.106,157.912
C07904=1046.029,343.728,-118.098,172.865,41.102,157.911
C07905=1046.021,343.482,-118.061,172.860,41.098,157.910
C07906=1046.014,343.234,-118.024,172.856,41.094,157.909
C07907=1046.006,342.986,-117.988,172.850,41.091,157.908
C07908=1045.999,342.740,-117.951,172.846,41.087,157.907
C07909=1045.992,342.492,-117.914,172.841,41.083,157.906
C07910=1045.985,342.245,-117.878,172.837,41.079,157.904
C07911=1045.977,341.998,-117.840,172.831,41.075,157.903
C07912=1045.970,341.751,-117.805,172.827,41.072,157.902
C07913=1045.963,341.503,-117.768,172.822,41.068,157.901
C07914=1045.956,341.256,-117.732,172.817,41.064,157.900
C07915=1045.949,341.009,-117.696,172.812,41.061,157.899
C07916=1045.941,340.761,-117.660,172.807,41.057,157.898
C07917=1045.934,340.514,-117.622,172.803,41.053,157.897
C07918=1045.927,340.268,-117.586,172.798,41.050,157.895
C07919=1045.919,340.020,-117.550,172.793,41.046,157.894
C07920=1045.912,339.772,-117.513,172.789,41.043,157.893
C07921=1045.905,339.526,-117.477,172.784,41.039,157.892
C07922=1045.897,339.278,-117.441,172.780,41.036,157.891
C07923=1045.891,339.031,-117.405,172.775,41.032,157.890
C07924=1045.883,338.784,-117.368,172.770,41.028,157.889
C07925=1045.876,338.536,-117.332,172.765,41.025,157.888
C07926=1045.869,338.290,-117.296,172.761,41.021,157.887
C07927=1045.862,338.041,-117.260,172.756,41.017,157.886
C07928=1045.855,337.794,-117.224,172.752,41.014,157.885
C07929=1045.847,337.547,-117.188,172.747,41.010,157.884
C07930=1045.841,337.300,-117.152,172.742,41.007,157.883
C07931=1045.833,337.052,-117.115,172.738,41.003,157.881
C07932=1045.826,336.806,-117.080,172.733,40.999,157.880
C07933=1045.819,336.558,-117.043,172.729,40.996,157.879
C07934=1045.812,336.311,-117.008,172.724,40.992,157.878
C07935=1045.805,336.063,-116.971,172.719,40.989,157.877
C07936=1045.798,335.816,-116.936,172.715,40.985,157.876
C07937=1045.791,335.568,-116.900,172.710,40.982,157.875
C07938=1045.784,335.321,-116.864,172.706,40.978,157.874
C07939=1045.776,335.074,-116.827,172.701,40.975,157.873
C07940=1045.770,334.826,-116.792,172.697,40.971,157.872
C07941=1045.762,334.579,-116.756,172.692,40.968,157.871
C07942=1045.755,334.332,-116.721,172.687,40.965,157.870
C07943=1045.747,334.084,-116.685,172.683,40.961,157.869
C07944=1045.738,333.768,-116.639,172.678,40.957,157.868
C07945=1045.729,333.450,-116.593,172.671,40.952,157.866
C07946=1045.721,333.134,-116.547,172.666,40.948,157.865
C07947=1045.711,332.816,-116.502,172.660,40.943,157.864
C07948=1045.703,332.569,-116.466,172.655,40.940,157.863
C07949=1045.697,332.322,-116.431,172.651,40.937,157.862
C07950=1045.690,332.075,-116.395,172.647,40.933,157.861
C07951=1045.682,331.827,-116.360,172.642,40.930,157.860
C07952=1045.675,331.579,-116.325,172.638,40.926,157.859
C07953=1045.668,331.332,-116.288,172.634,40.923,157.858
C07954=1045.661,331.085,-116.253,172.629,40.919,157.857
C07955=1045.654,330.837,-116.218,172.624,40.916,157.856
C07956=1045.647,330.590,-116.182,172.620,40.913,157.855
C07957=1045.640,330.342,-116.147,172.616,40.909,157.854
C07958=1045.633,330.095,-116.112,172.611,40.906,157.853
C07959=1045.626,329.848,-116.076,172.607,40.902,157.852
C07960=1045.619,329.601,-116.041,172.603,40.899,157.851
C07961=1045.612,329.353,-116.005,172.599,40.896,157.850
C07962=1045.605,329.105,-115.970,172.594,40.893,157.849
C07963=1045.598,328.858,-115.935,172.590,40.889,157.848
C07964=1045.590,328.610,-115.900,172.586,40.886,157.847
C07965=1045.583,328.363,-115.865,172.581,40.883,157.846
C07966=1045.577,328.116,-115.830,172.577,40.880,157.845
C07967=1045.569,327.868,-115.795,172.573,40.876,157.844
C07968=1045.562,327.620,-115.760,172.569,40.873,157.843
C07969=1045.554,327.373,-115.725,172.563,40.870,157.842
C07970=1045.548,327.126,-115.690,172.559,40.866,157.841
C07971=1045.540,326.878,-115.654,172.555,40.863,157.840
C07972=1045.533,326.631,-115.620,172.551,40.860,157.839
C07973=1045.526,326.384,-115.585,172.546,40.857,157.838
C07974=1045.518,326.137,-115.550,172.542,40.854,157.837
C07975=1045.512,325.889,-115.516,172.538,40.851,157.836
C07976=1045.505,325.640,-115.480,172.534,40.847,157.835
C07977=1045.497,325.393,-115.446,172.529,40.844,157.834
C07978=1045.490,325.146,-115.411,172.525,40.841,157.833
C07979=1045.483,324.899,-115.376,172.521,40.838,157.833
C07980=1045.476,324.652,-115.341,172.517,40.835,157.832
C07981=1045.470,324.404,-115.307,172.513,40.832,157.831
C07982=1045.461,324.156,-115.272,172.508,40.828,157.830
C07983=1045.455,323.909,-115.237,172.504,40.825,157.829
C07984=1045.447,323.661,-115.202,172.500,40.822,157.828
C07985=1045.441,323.413,-115.168,172.496,40.819,157.827
C07986=1045.434,323.166,-115.132,172.492,40.816,157.826
C07987=1045.426,322.919,-115.098,172.487,40.813,157.825
C07988=1045.420,322.671,-115.063,172.483,40.809,157.824
C07989=1045.412,322.424,-115.029,172.479,40.806,157.823
C07990=1045.406,322.176,-114.995,172.475,40.803,157.822
C07991=1045.398,321.929,-114.960,172.471,40.800,157.821
C07992=1045.392,321.682,-114.925,172.467,40.797,157.820
C07993=1045.385,321.434,-114.891,172.463,40.793,157.819
C07994=1045.378,321.187,-114.856,172.458,40.791,157.819
C07995=1045.371,320.939,-114.821,172.454,40.788,157.818
C07996=1045.364,320.692,-114.787,172.450,40.784,157.817
C07997=1045.357,320.444,-114.752,172.446,40.781,157.816
C07998=1045.350,320.197,-114.718,172.442,40.778,157.815
C07999=1045.343,319.949,-114.684,172.438,40.775,157.814
C08000=1045.334,319.627,-114.639,172.433,40.771,157.813
C08001=1045.325,319.305,-114.594,172.427,40.767,157.812
C08002=1045.316,318.982,-114.549,172.422,40.763,157.810
C08003=1045.307,318.661,-114.505,172.417,40.759,157.809
C08004=1045.300,318.413,-114.470,172.413,40.756,157.808
C08005=1045.293,318.166,-114.436,172.409,40.752,157.807
C08006=1045.286,317.918,-114.401,172.405,40.749,157.807
C08007=1045.280,317.671,-114.368,172.401,40.747,157.806
C08008=1045.273,317.423,-114.333,172.396,40.744,157.805
C08009=1045.266,317.176,-114.299,172.392,40.740,157.804
C08010=1045.259,316.928,-114.265,172.388,40.737,157.803
C08011=1045.253,316.680,-114.229,172.384,40.734,157.802
C08012=1045.245,316.433,-114.196,172.380,40.731,157.801
C08013=1045.239,316.186,-114.162,172.376,40.728,157.800
C08014=1045.232,315.938,-114.128,172.372,40.725,157.799
C08015=1045.225,315.690,-114.094,172.368,40.722,157.799
C08016=1045.218,315.443,-114.059,172.364,40.719,157.798
C08017=1045.212,315.196,-114.025,172.360,40.716,157.797
C08018=1045.205,314.948,-113.991,172.356,40.713,157.796
C08019=1045.198,314.700,-113.957,172.352,40.710,157.795
C08020=1045.192,314.452,-113.923,172.348,40.707,157.794
C08021=1045.185,314.205,-113.889,172.344,40.704,157.793
C08022=1045.179,313.957,-113.855,172.340,40.701,157.792
C08023=1045.171,313.709,-113.821,172.336,40.698,157.792
C08024=1045.166,313.462,-113.787,172.333,40.695,157.791
C08025=1045.158,313.215,-113.752,172.329,40.692,157.790
C08026=1045.152,312.967,-113.718,172.325,40.688,157.789
C08027=1045.145,312.720,-113.684,172.321,40.686,157.788
C08028=1045.138,312.472,-113.651,172.317,40.683,157.787
C08029=1045.131,312.224,-113.618,172.313,40.680,157.786
C08030=1045.124,311.976,-113.584,172.309,40.677,157.786
C08031=1045.117,311.729,-113.550,172.305,40.674,157.785
C08032=1045.110,311.482,-113.516,172.301,40.671,157.784
C08033=1045.103,311.234,-113.483,172.297,40.668,157.783
C08034=1045.096,310.986,-113.450,172.293,40.666,157.782
C08035=1045.089,310.739,-113.416,172.290,40.663,157.782
C08036=1045.082,310.491,-113.382,172.286,40.660,157.781
C08037=1045.075,310.243,-113.349,172.282,40.657,157.780
C08038=1045.068,309.995,-113.315,172.278,40.654,157.779
C08039=1045.061,309.749,-113.282,172.275,40.651,157.778
C08040=1045.054,309.500,-113.249,172.271,40.648,157.777
C08041=1045.046,309.253,-113.215,172.267,40.646,157.777
C08042=1045.040,309.006,-113.182,172.263,40.643,157.776
C08043=1045.033,308.757,-113.149,172.259,40.640,157.775
C08044=1045.026,308.510,-113.115,172.256,40.637,157.774
C08045=1045.020,308.262,-113.082,172.252,40.634,157.773
C08046=1045.012,308.014,-113.049,172.248,40.631,157.772
C08047=1045.006,307.767,-113.015,172.244,40.629,157.772
C08048=1044.998,307.519,-112.983,172.240,40.626,157.771
C08049=1044.991,307.272,-112.949,172.236,40.623,157.770
C08050=1044.985,307.024,-112.916,172.232,40.620,157.769
C08051=1044.977,306.776,-112.882,172.228,40.618,157.768
C08052=1044.971,306.529,-112.849,172.225,40.615,157.768
C08053=1044.964,306.281,-112.816,172.221,40.612,157.767
C08054=1044.958,306.034,-112.783,172.218,40.609,157.766
C08055=1044.950,305.786,-112.750,172.214,40.606,157.765
C08056=1044.941,305.468,-112.708,172.209,40.603,157.764
C08057=1044.933,305.151,-112.665,172.204,40.599,157.763
C08058=1044.924,304.834,-112.623,172.200,40.596,157.762
C08059=1044.915,304.516,-112.580,172.194,40.592,157.761
C08060=1044.908,304.269,-112.547,172.191,40.589,157.760
C08061=1044.901,304.021,-112.514,172.187,40.587,157.760
C08062=1044.895,303.773,-112.481,172.183,40.584,157.759
C08063=1044.889,303.526,-112.448,172.179,40.581,157.758
C08064=1044.882,303.277,-112.415,172.176,40.578,157.757
C08065=1044.874,303.031,-112.382,172.172,40.575,157.756
C08066=1044.868,302.783,-112.349,172.169,40.573,157.756
C08067=1044.861,302.535,-112.316,172.165,40.570,157.755
C08068=1044.854,302.287,-112.283,172.161,40.567,157.754
C08069=1044.848,302.040,-112.250,172.157,40.565,157.753
C08070=1044.841,301.792,-112.217,172.154,40.561,157.752
C08071=1044.834,301.544,-112.184,172.150,40.559,157.752
C08072=1044.828,301.296,-112.152,172.146,40.556,157.751
C08073=1044.821,301.048,-112.119,172.143,40.553,157.750
C08074=1044.814,300.801,-112.086,172.139,40.551,157.749
C08075=1044.808,300.554,-112.052,172.136,40.548,157.748
C08076=1044.801,300.305,-112.019,172.132,40.545,157.748
C08077=1044.794,300.058,-111.987,172.128,40.543,157.747
C08078=1044.788,299.810,-111.954,172.125,40.540,157.746
C08079=1044.781,299.563,-111.922,172.122,40.536,157.745
C08080=1044.774,299.315,-111.889,172.118,40.534,157.745
C08081=1044.768,299.067,-111.856,172.114,40.531,157.744
C08082=1044.761,298.820,-111.824,172.110,40.528,157.743
C08083=1044.754,298.571,-111.791,172.107,40.526,157.742
C08084=1044.748,298.324,-111.758,172.104,40.523,157.741
C08085=1044.742,298.076,-111.725,172.100,40.520,157.741
C08086=1044.735,297.829,-111.693,172.096,40.518,157.740
C08087=1044.728,297.581,-111.660,172.093,40.515,157.739
C08088=1044.721,297.333,-111.627,172.089,40.512,157.738
C08089=1044.715,297.085,-111.594,172.085,40.510,157.738
C08090=1044.709,296.838,-111.562,172.082,40.507,157.737
C08091=1044.701,296.589,-111.530,172.079,40.504,157.736
C08092=1044.695,296.342,-111.497,172.075,40.501,157.735
C08093=1044.689,296.094,-111.464,172.071,40.499,157.735
C08094=1044.683,295.846,-111.432,172.068,40.496,157.734
C08095=1044.676,295.599,-111.399,172.065,40.493,157.733
C08096=1044.669,295.350,-111.367,172.061,40.491,157.732
C08097=1044.662,295.103,-111.335,172.057,40.488,157.732
C08098=1044.656,294.855,-111.302,172.054,40.485,157.731
C08099=1044.649,294.608,-111.270,172.050,40.483,157.730
C08100=1044.642,294.359,-111.238,172.046,40.480,157.729
C08101=1044.635,294.112,-111.205,172.044,40.477,157.729
C08102=1044.629,293.864,-111.173,172.040,40.475,157.728
C08103=1044.622,293.616,-111.141,172.036,40.472,157.727
C08104=1044.615,293.369,-111.109,172.032,40.470,157.726
C08105=1044.608,293.120,-111.077,172.030,40.467,157.726
C08106=1044.601,292.873,-111.045,172.026,40.464,157.725
C08107=1044.595,292.625,-111.013,172.022,40.462,157.724
C08108=1044.588,292.377,-110.980,172.019,40.459,157.723
C08109=1044.582,292.130,-110.949,172.016,40.457,157.723
C08110=1044.575,291.882,-110.917,172.012,40.454,157.722
C08111=1044.568,291.633,-110.884,172.009,40.452,157.721
C08112=1044.560,291.333,-110.845,172.004,40.449,157.720
C08113=1044.551,291.031,-110.807,172.000,40.445,157.720
C08114=1044.543,290.731,-110.768,171.996,40.442,157.719
C08115=1044.535,290.430,-110.729,171.992,40.439,157.718
C08116=1044.529,290.182,-110.697,171.989,40.437,157.717
C08117=1044.522,289.934,-110.665,171.985,40.434,157.716
C08118=1044.515,289.686,-110.633,171.982,40.431,157.716
C08119=1044.509,289.438,-110.601,171.978,40.429,157.715
C08120=1044.502,289.190,-110.569,171.975,40.426,157.714
C08121=1044.495,288.943,-110.538,171.972,40.424,157.713
C08122=1044.488,288.695,-110.506,171.968,40.421,157.713
C08123=1044.482,288.447,-110.474,171.965,40.419,157.712
C08124=1044.475,288.199,-110.442,171.961,40.416,157.711
C08125=1044.469,287.951,-110.411,171.958,40.413,157.711
C08126=1044.462,287.703,-110.379,171.955,40.411,157.710
C08127=1044.456,287.456,-110.347,171.951,40.409,157.709
C08128=1044.449,287.208,-110.315,171.948,40.406,157.708
C08129=1044.442,286.960,-110.284,171.945,40.404,157.708
C08130=1044.435,286.711,-110.252,171.941,40.401,157.707
C08131=1044.428,286.463,-110.220,171.938,40.398,157.706
C08132=1044.421,286.215,-110.189,171.934,40.396,157.706
C08133=1044.414,285.968,-110.157,171.932,40.393,157.705
C08134=1044.408,285.720,-110.125,171.928,40.391,157.704
C08135=1044.401,285.472,-110.094,171.924,40.389,157.704
C08136=1044.394,285.225,-110.063,171.922,40.386,157.703
C08137=1044.387,284.977,-110.031,171.918,40.384,157.702
C08138=1044.381,284.729,-110.000,171.915,40.381,157.701
C08139=1044.374,284.481,-109.968,171.911,40.379,157.701
C08140=1044.367,284.233,-109.937,171.908,40.376,157.700
C08141=1044.361,283.985,-109.905,171.905,40.374,157.699
C08142=1044.354,283.737,-109.874,171.901,40.371,157.699
C08143=1044.347,283.489,-109.843,171.899,40.369,157.698
C08144=1044.340,283.241,-109.811,171.895,40.366,157.697
C08145=1044.334,282.993,-109.780,171.892,40.364,157.697
C08146=1044.327,282.745,-109.748,171.888,40.361,157.696
C08147=1044.320,282.497,-109.718,171.885,40.359,157.695
C08148=1044.314,282.250,-109.686,171.882,40.356,157.695
C08149=1044.308,282.002,-109.655,171.879,40.354,157.694
C08150=1044.301,281.754,-109.624,171.875,40.352,157.693
C08151=1044.294,281.506,-109.592,171.872,40.349,157.693
C08152=1044.287,281.258,-109.561,171.869,40.347,157.692
C08153=1044.281,281.010,-109.529,171.865,40.344,157.691
C08154=1044.274,280.762,-109.499,171.863,40.342,157.691
C08155=1044.268,280.514,-109.467,171.859,40.339,157.690
C08156=1044.261,280.266,-109.436,171.856,40.337,157.689
C08157=1044.255,280.019,-109.405,171.852,40.334,157.688
C08158=1044.248,279.771,-109.373,171.850,40.332,157.688
C08159=1044.242,279.522,-109.342,171.846,40.329,157.687
C08160=1044.235,279.274,-109.311,171.843,40.327,157.687
C08161=1044.228,279.026,-109.280,171.840,40.324,157.686
C08162=1044.222,278.778,-109.249,171.837,40.322,157.685
C08163=1044.215,278.530,-109.217,171.834,40.319,157.684
C08164=1044.209,278.283,-109.186,171.830,40.317,157.684
C08165=1044.202,278.034,-109.156,171.828,40.314,157.683
C08166=1044.195,277.787,-109.125,171.824,40.312,157.682
C08167=1044.188,277.539,-109.093,171.821,40.310,157.682
C08168=1044.181,277.249,-109.058,171.817,40.307,157.681
C08169=1044.173,276.960,-109.021,171.814,40.304,157.680
C08170=1044.165,276.670,-108.986,171.810,40.301,157.679
C08171=1044.157,276.381,-108.950,171.806,40.299,157.679
C08172=1044.151,276.133,-108.919,171.803,40.296,157.678
C08173=1044.144,275.885,-108.888,171.800,40.294,157.677
C08174=1044.138,275.636,-108.857,171.797,40.292,157.677
C08175=1044.130,275.389,-108.826,171.793,40.289,157.676
C08176=1044.124,275.141,-108.796,171.791,40.287,157.675
C08177=1044.118,274.893,-108.764,171.787,40.285,157.675
C08178=1044.111,274.645,-108.734,171.784,40.282,157.674
C08179=1044.104,274.397,-108.703,171.782,40.280,157.673
C08180=1044.098,274.149,-108.672,171.778,40.277,157.673
C08181=1044.092,273.901,-108.642,171.775,40.275,157.672
C08182=1044.084,273.653,-108.611,171.771,40.272,157.671
C08183=1044.078,273.405,-108.580,171.769,40.270,157.671
C08184=1044.072,273.157,-108.549,171.765,40.268,157.670
C08185=1044.064,272.909,-108.519,171.762,40.265,157.670
C08186=1044.058,272.661,-108.488,171.760,40.263,157.669
C08187=1044.051,272.413,-108.457,171.756,40.260,157.668
C08188=1044.045,272.165,-108.427,171.753,40.258,157.668
C08189=1044.038,271.917,-108.396,171.750,40.256,157.667
C08190=1044.032,271.668,-108.366,171.747,40.253,157.666
C08191=1044.025,271.421,-108.335,171.744,40.251,157.666
C08192=1044.019,271.173,-108.304,171.741,40.249,157.665
C08193=1044.012,270.925,-108.274,171.738,40.247,157.664
C08194=1044.006,270.677,-108.244,171.735,40.244,157.664
C08195=1043.999,270.429,-108.214,171.732,40.242,157.663
C08196=1043.992,270.180,-108.183,171.729,40.240,157.662
C08197=1043.985,269.932,-108.152,171.725,40.237,157.662
C08198=1043.979,269.685,-108.122,171.723,40.235,157.661
C08199=1043.972,269.436,-108.092,171.720,40.232,157.661
C08200=1043.965,269.188,-108.061,171.716,40.230,157.660
C08201=1043.959,268.940,-108.031,171.714,40.227,157.659
C08202=1043.952,268.692,-108.001,171.711,40.225,157.659
C08203=1043.946,268.444,-107.971,171.707,40.223,157.658
C08204=1043.939,268.196,-107.940,171.705,40.221,157.657
C08205=1043.932,267.948,-107.910,171.702,40.219,157.657
C08206=1043.926,267.700,-107.880,171.698,40.216,157.656
C08207=1043.919,267.452,-107.850,171.696,40.214,157.655
C08208=1043.912,267.203,-107.819,171.692,40.212,157.655
C08209=1043.906,266.955,-107.789,171.689,40.209,157.654
C08210=1043.899,266.707,-107.759,171.687,40.207,157.654
C08211=1043.892,266.460,-107.729,171.683,40.204,157.653
C08212=1043.886,266.211,-107.698,171.680,40.202,157.652
C08213=1043.879,265.963,-107.668,171.678,40.200,157.652
C08214=1043.872,265.716,-107.639,171.675,40.198,157.651
C08215=1043.866,265.467,-107.608,171.672,40.196,157.651
C08216=1043.859,265.219,-107.578,171.669,40.193,157.650
C08217=1043.853,264.971,-107.549,171.666,40.191,157.649
C08218=1043.847,264.723,-107.518,171.663,40.188,157.649
C08219=1043.840,264.475,-107.488,171.660,40.186,157.648
C08220=1043.832,264.226,-107.458,171.657,40.184,157.647
C08221=1043.827,263.979,-107.428,171.654,40.182,157.647
C08222=1043.819,263.730,-107.398,171.651,40.179,157.646
C08223=1043.813,263.482,-107.369,171.648,40.177,157.645
C08224=1043.805,263.198,-107.333,171.645,40.174,157.645
C08225=1043.798,262.913,-107.299,171.642,40.172,157.644
C08226=1043.791,262.628,-107.265,171.638,40.169,157.643
C08227=1043.783,262.342,-107.230,171.634,40.166,157.643
C08228=1043.777,262.095,-107.200,171.632,40.164,157.642
C08229=1043.770,261.846,-107.171,171.629,40.162,157.641
C08230=1043.763,261.598,-107.141,171.627,40.160,157.641
C08231=1043.756,261.350,-107.112,171.623,40.158,157.640
C08232=1043.749,261.102,-107.082,171.620,40.155,157.640
C08233=1043.743,260.854,-107.052,171.618,40.153,157.639
C08234=1043.736,260.605,-107.023,171.614,40.151,157.638
C08235=1043.729,260.358,-106.993,171.611,40.149,157.638
C08236=1043.722,260.109,-106.963,171.609,40.147,157.637
C08237=1043.716,259.861,-106.934,171.606,40.144,157.637
C08238=1043.709,259.612,-106.904,171.603,40.142,157.636
C08239=1043.702,259.365,-106.875,171.600,40.140,157.635
C08240=1043.696,259.116,-106.845,171.597,40.138,157.635
C08241=1043.688,258.869,-106.816,171.595,40.135,157.634
C08242=1043.681,258.620,-106.787,171.591,40.133,157.634
C08243=1043.675,258.373,-106.757,171.589,40.131,157.633
C08244=1043.668,258.124,-106.727,171.586,40.129,157.633
C08245=1043.662,257.876,-106.698,171.583,40.127,157.632
C08246=1043.655,257.627,-106.668,171.580,40.125,157.631
C08247=1043.648,257.379,-106.639,171.577,40.122,157.631
C08248=1043.641,257.131,-106.609,171.574,40.120,157.630
C08249=1043.635,256.883,-106.580,171.572,40.118,157.630
C08250=1043.628,256.634,-106.551,171.568,40.116,157.629
C08251=1043.622,256.387,-106.521,171.566,40.113,157.628
C08252=1043.615,256.138,-106.492,171.563,40.111,157.628
C08253=1043.608,255.890,-106.462,171.560,40.109,157.627
C08254=1043.602,255.642,-106.433,171.558,40.107,157.627
C08255=1043.595,255.393,-106.403,171.554,40.105,157.626
C08256=1043.588,255.145,-106.375,171.552,40.102,157.625
C08257=1043.581,254.898,-106.345,171.549,40.100,157.625
C08258=1043.575,254.649,-106.316,171.546,40.098,157.624
C08259=1043.568,254.401,-106.287,171.544,40.096,157.624
C08260=1043.562,254.153,-106.258,171.540,40.094,157.623
C08261=1043.555,253.905,-106.227,171.538,40.091,157.622
C08262=1043.549,253.657,-106.198,171.535,40.089,157.622
C08263=1043.542,253.408,-106.169,171.532,40.087,157.621
C08264=1043.536,253.160,-106.140,171.530,40.085,157.621
C08265=1043.529,252.912,-106.110,171.527,40.082,157.620
C08266=1043.523,252.664,-106.081,171.524,40.079,157.619
C08267=1043.515,252.415,-106.052,171.521,40.077,157.619
C08268=1043.509,252.167,-106.023,171.518,40.075,157.618
C08269=1043.503,251.919,-105.994,171.515,40.073,157.618
C08270=1043.496,251.670,-105.965,171.513,40.071,157.617
C08271=1043.490,251.422,-105.936,171.510,40.068,157.616
C08272=1043.483,251.175,-105.906,171.508,40.066,157.616
C08273=1043.476,250.926,-105.877,171.505,40.064,157.615
C08274=1043.470,250.678,-105.848,171.501,40.062,157.615
C08275=1043.464,250.430,-105.819,171.499,40.059,157.614
C08276=1043.457,250.182,-105.790,171.496,40.057,157.613
C08277=1043.450,249.933,-105.761,171.494,40.055,157.613
C08278=1043.444,249.685,-105.732,171.491,40.053,157.612
C08279=1043.437,249.437,-105.703,171.488,40.050,157.612
C08280=1043.430,249.150,-105.669,171.486,40.048,157.611
C08281=1043.423,248.864,-105.636,171.482,40.045,157.610
C08282=1043.415,248.577,-105.602,171.479,40.043,157.610
C08283=1043.408,248.291,-105.569,171.476,40.040,157.609
C08284=1043.401,248.042,-105.540,171.473,40.038,157.608
C08285=1043.394,247.794,-105.511,171.470,40.036,157.608
C08286=1043.388,247.546,-105.482,171.468,40.033,157.607
C08287=1043.382,247.298,-105.453,171.465,40.031,157.607
C08288=1043.376,247.050,-105.424,171.463,40.029,157.606
C08289=1043.370,246.802,-105.395,171.460,40.026,157.605
C08290=1043.362,246.553,-105.366,171.457,40.024,157.605
C08291=1043.356,246.305,-105.337,171.455,40.022,157.604
C08292=1043.349,246.057,-105.308,171.452,40.020,157.604
C08293=1043.343,245.809,-105.279,171.450,40.017,157.603
C08294=1043.337,245.561,-105.250,171.447,40.015,157.602
C08295=1043.331,245.312,-105.221,171.444,40.013,157.602
C08296=1043.323,245.063,-105.192,171.442,40.011,157.601
C08297=1043.317,244.815,-105.163,171.439,40.008,157.601
C08298=1043.310,244.568,-105.135,171.437,40.006,157.600
C08299=1043.304,244.319,-105.107,171.434,40.004,157.600
C08300=1043.298,244.071,-105.078,171.430,40.002,157.599
C08301=1043.291,243.823,-105.049,171.428,39.999,157.598
C08302=1043.285,243.575,-105.020,171.425,39.998,157.598
C08303=1043.277,243.326,-104.992,171.423,39.996,157.597
C08304=1043.271,243.077,-104.963,171.420,39.993,157.597
C08305=1043.265,242.829,-104.934,171.417,39.991,157.596
C08306=1043.258,242.581,-104.906,171.415,39.989,157.596
C08307=1043.252,242.333,-104.877,171.412,39.987,157.595
C08308=1043.245,242.085,-104.849,171.410,39.984,157.594
C08309=1043.239,241.836,-104.820,171.407,39.982,157.594
C08310=1043.233,241.588,-104.791,171.404,39.980,157.593
C08311=1043.226,241.340,-104.763,171.402,39.978,157.593
C08312=1043.219,241.091,-104.734,171.399,39.975,157.592
C08313=1043.212,240.843,-104.706,171.397,39.973,157.592
C08314=1043.206,240.594,-104.678,171.394,39.971,157.591
C08315=1043.199,240.346,-104.649,171.391,39.969,157.590
C08316=1043.193,240.098,-104.621,171.389,39.967,157.590
C08317=1043.186,239.850,-104.593,171.386,39.965,157.589
C08318=1043.180,239.601,-104.564,171.384,39.962,157.589
C08319=1043.173,239.354,-104.536,171.381,39.960,157.588
C08320=1043.167,239.105,-104.508,171.379,39.958,157.588
C08321=1043.159,238.856,-104.479,171.376,39.956,157.587
C08322=1043.153,238.608,-104.451,171.373,39.953,157.586
C08323=1043.146,238.360,-104.422,171.371,39.952,157.586
C08324=1043.140,238.111,-104.394,171.368,39.949,157.585
C08325=1043.133,237.863,-104.367,171.366,39.947,157.585
C08326=1043.127,237.615,-104.338,171.363,39.945,157.584
C08327=1043.120,237.366,-104.310,171.361,39.943,157.584
C08328=1043.113,237.118,-104.282,171.358,39.940,157.583
C08329=1043.106,236.870,-104.254,171.355,39.938,157.582
C08330=1043.100,236.621,-104.225,171.354,39.936,157.582
C08331=1043.094,236.373,-104.198,171.351,39.934,157.581
C08332=1043.087,236.125,-104.169,171.349,39.932,157.581
C08333=1043.080,235.876,-104.141,171.346,39.930,157.580
C08334=1043.074,235.628,-104.113,171.344,39.927,157.580
C08335=1043.067,235.380,-104.085,171.341,39.925,157.579
C08336=1043.059,235.087,-104.052,171.338,39.923,157.579
C08337=1043.051,234.795,-104.019,171.335,39.920,157.578
C08338=1043.044,234.503,-103.985,171.332,39.918,157.577
C08339=1043.036,234.211,-103.953,171.329,39.915,157.577
C08340=1043.029,233.963,-103.924,171.327,39.913,157.576
C08341=1043.023,233.714,-103.897,171.324,39.910,157.575
C08342=1043.017,233.466,-103.868,171.322,39.908,157.575
C08343=1043.010,233.217,-103.841,171.319,39.906,157.574
C08344=1043.004,232.969,-103.813,171.317,39.904,157.574
C08345=1042.997,232.721,-103.784,171.314,39.902,157.573
C08346=1042.991,232.472,-103.756,171.311,39.900,157.573
C08347=1042.984,232.224,-103.728,171.309,39.897,157.572
C08348=1042.977,231.975,-103.701,171.307,39.895,157.571
C08349=1042.971,231.727,-103.673,171.305,39.893,157.571
C08350=1042.964,231.479,-103.646,171.302,39.891,157.570
C08351=1042.958,231.231,-103.618,171.300,39.889,157.570
C08352=1042.952,230.982,-103.590,171.297,39.887,157.569
C08353=1042.945,230.734,-103.561,171.294,39.884,157.569
C08354=1042.938,230.486,-103.533,171.292,39.882,157.568
C08355=1042.931,230.237,-103.506,171.289,39.880,157.568
C08356=1042.925,229.989,-103.478,171.288,39.877,157.567
C08357=1042.918,229.740,-103.450,171.285,39.875,157.566
C08358=1042.911,229.492,-103.422,171.283,39.874,157.566
C08359=1042.905,229.243,-103.395,171.280,39.871,157.565
C08360=1042.898,228.995,-103.367,171.277,39.869,157.565
C08361=1042.892,228.747,-103.340,171.275,39.867,157.564
C08362=1042.886,228.498,-103.311,171.272,39.864,157.564
C08363=1042.879,228.250,-103.284,171.270,39.862,157.563
C08364=1042.872,228.001,-103.257,171.268,39.860,157.563
C08365=1042.866,227.753,-103.229,171.266,39.858,157.562
C08366=1042.859,227.504,-103.202,171.263,39.856,157.562
C08367=1042.852,227.256,-103.174,171.260,39.854,157.561
C08368=1042.846,227.007,-103.146,171.258,39.852,157.561
C08369=1042.839,226.759,-103.118,171.255,39.850,157.560
C08370=1042.833,226.511,-103.091,171.253,39.847,157.559
C08371=1042.826,226.262,-103.064,171.251,39.845,157.559
C08372=1042.819,226.014,-103.037,171.249,39.843,157.558
C08373=1042.812,225.766,-103.009,171.246,39.841,157.558
C08374=1042.806,225.517,-102.982,171.244,39.839,157.557
C08375=1042.799,225.269,-102.954,171.241,39.837,157.557
C08376=1042.792,225.020,-102.926,171.238,39.834,157.556
C08377=1042.786,224.772,-102.899,171.237,39.832,157.555
C08378=1042.780,224.524,-102.872,171.234,39.830,157.555
C08379=1042.772,224.275,-102.845,171.232,39.828,157.554
C08380=1042.766,224.027,-102.817,171.229,39.826,157.554
C08381=1042.759,223.778,-102.790,171.227,39.823,157.553
C08382=1042.753,223.530,-102.762,171.225,39.821,157.553
C08383=1042.747,223.282,-102.735,171.223,39.819,157.552
C08384=1042.740,223.033,-102.708,171.220,39.817,157.552
C08385=1042.734,222.784,-102.680,171.218,39.815,157.551
C08386=1042.727,222.536,-102.652,171.215,39.813,157.551
C08387=1042.720,222.288,-102.625,171.213,39.810,157.550
C08388=1042.714,222.039,-102.598,171.211,39.808,157.549
C08389=1042.707,221.791,-102.571,171.208,39.806,157.549
C08390=1042.701,221.542,-102.544,171.206,39.804,157.548
C08391=1042.694,221.294,-102.516,171.204,39.802,157.548
C08392=1042.686,220.995,-102.484,171.201,39.799,157.547
C08393=1042.678,220.695,-102.451,171.198,39.796,157.546
C08394=1042.671,220.395,-102.418,171.195,39.794,157.546
C08395=1042.662,220.095,-102.385,171.192,39.791,157.545
C08396=1042.656,219.847,-102.358,171.190,39.789,157.545
C08397=1042.649,219.599,-102.331,171.188,39.787,157.544
C08398=1042.643,219.350,-102.304,171.186,39.784,157.544
C08399=1042.636,219.101,-102.276,171.183,39.782,157.543
C08400=1042.629,218.853,-102.250,171.181,39.780,157.542
C08401=1042.623,218.605,-102.222,171.179,39.778,157.542
C08402=1042.616,218.356,-102.196,171.177,39.776,157.541
C08403=1042.609,218.108,-102.168,171.174,39.774,157.541
C08404=1042.602,217.859,-102.142,171.172,39.771,157.540
C08405=1042.596,217.610,-102.115,171.170,39.770,157.540
C08406=1042.589,217.362,-102.087,171.168,39.767,157.539
C08407=1042.583,217.114,-102.061,171.165,39.765,157.539
C08408=1042.576,216.865,-102.033,171.162,39.763,157.538
C08409=1042.569,216.617,-102.007,171.161,39.760,157.538
C08410=1042.562,216.368,-101.979,171.158,39.759,157.537
C08411=1042.557,216.120,-101.953,171.156,39.756,157.537
C08412=1042.549,215.871,-101.926,171.154,39.754,157.536
C08413=1042.543,215.623,-101.899,171.152,39.752,157.535
C08414=1042.536,215.375,-101.872,171.149,39.749,157.535
C08415=1042.530,215.126,-101.845,171.147,39.748,157.534
C08416=1042.522,214.878,-101.818,171.145,39.745,157.534
C08417=1042.517,214.629,-101.792,171.143,39.743,157.533
C08418=1042.510,214.380,-101.765,171.140,39.741,157.533
C08419=1042.503,214.133,-101.738,171.138,39.738,157.532
C08420=1042.497,213.884,-101.711,171.136,39.736,157.532
C08421=1042.490,213.635,-101.684,171.133,39.735,157.531
C08422=1042.484,213.386,-101.658,171.132,39.732,157.531
C08423=1042.477,213.138,-101.631,171.129,39.730,157.530
C08424=1042.470,212.889,-101.604,171.127,39.728,157.529
C08425=1042.464,212.641,-101.578,171.125,39.725,157.529
C08426=1042.458,212.392,-101.551,171.123,39.723,157.528
C08427=1042.451,212.145,-101.524,171.120,39.721,157.528
C08428=1042.444,211.896,-101.497,171.119,39.719,157.527
C08429=1042.438,211.648,-101.471,171.116,39.717,157.527
C08430=1042.431,211.399,-101.444,171.113,39.714,157.526
C08431=1042.424,211.150,-101.417,171.112,39.712,157.526
C08432=1042.418,210.902,-101.390,171.109,39.710,157.525
C08433=1042.411,210.653,-101.364,171.107,39.708,157.525
C08434=1042.405,210.405,-101.337,171.105,39.706,157.524
C08435=1042.398,210.156,-101.310,171.103,39.703,157.524
C08436=1042.391,209.907,-101.284,171.100,39.701,157.523
C08437=1042.385,209.659,-101.257,171.099,39.699,157.522
C08438=1042.378,209.410,-101.231,171.096,39.697,157.522
C08439=1042.372,209.162,-101.205,171.094,39.695,157.521
C08440=1042.365,208.913,-101.178,171.092,39.692,157.521
C08441=1042.359,208.665,-101.152,171.089,39.690,157.520
C08442=1042.352,208.416,-101.125,171.088,39.688,157.520
C08443=1042.345,208.168,-101.099,171.085,39.686,157.519
C08444=1042.339,207.919,-101.072,171.083,39.684,157.519
C08445=1042.332,207.671,-101.046,171.081,39.681,157.518
C08446=1042.325,207.423,-101.020,171.079,39.679,157.518
C08447=1042.319,207.173,-100.993,171.076,39.677,157.517
C08448=1042.311,206.880,-100.962,171.075,39.674,157.516
C08449=1042.303,206.586,-100.930,171.072,39.672,157.516
C08450=1042.295,206.292,-100.900,171.069,39.669,157.515
C08451=1042.287,205.997,-100.868,171.067,39.667,157.515
C08452=1042.259,204.859,-100.753,170.790,39.564,157.484
C08453=1042.253,204.632,-100.730,170.787,39.563,157.483
C08454=1042.247,204.405,-100.707,170.785,39.561,157.483
C08455=1042.242,204.177,-100.684,170.782,39.560,157.483
C08456=1042.236,203.928,-100.659,170.779,39.558,157.482
C08457=1042.230,203.679,-100.634,170.777,39.556,157.482
C08458=1042.224,203.431,-100.608,170.773,39.555,157.481
C08459=1042.218,203.183,-100.583,170.771,39.554,157.481
C08460=1042.211,202.935,-100.559,170.767,39.552,157.480
C08461=1042.205,202.685,-100.534,170.764,39.551,157.480
C08462=1042.199,202.437,-100.509,170.762,39.549,157.480
C08463=1042.193,202.188,-100.483,170.758,39.548,157.479
C08464=1042.186,201.939,-100.458,170.756,39.547,157.479
C08465=1042.181,201.691,-100.434,170.753,39.545,157.479
C08466=1042.175,201.442,-100.408,170.750,39.544,157.478
C08467=1042.169,201.193,-100.383,170.747,39.542,157.478
C08468=1042.162,200.944,-100.359,170.744,39.541,157.477
C08469=1042.156,200.696,-100.334,170.741,39.540,157.477
C08470=1042.150,200.447,-100.308,170.739,39.539,157.477
C08471=1042.144,200.199,-100.285,170.735,39.537,157.476
C08472=1042.137,199.950,-100.259,170.733,39.536,157.476
C08473=1042.131,199.701,-100.235,170.730,39.534,157.476
C08474=1042.125,199.452,-100.210,170.727,39.533,157.475
C08475=1042.118,199.204,-100.185,170.724,39.532,157.475
C08476=1042.112,198.955,-100.161,170.722,39.531,157.475
C08477=1042.106,198.707,-100.136,170.718,39.529,157.474
C08478=1042.100,198.458,-100.112,170.715,39.528,157.474
C08479=1042.093,198.209,-100.086,170.713,39.527,157.473
C08480=1042.087,197.960,-100.062,170.709,39.525,157.473
C08481=1042.080,197.711,-100.037,170.707,39.524,157.473
C08482=1042.075,197.463,-100.013,170.704,39.523,157.472
C08483=1042.068,197.215,-99.988,170.701,39.521,157.472
C08484=1042.062,196.965,-99.963,170.698,39.520,157.472
C08485=1042.056,196.716,-99.939,170.696,39.519,157.471
C08486=1042.050,196.468,-99.914,170.692,39.518,157.471
C08487=1042.043,196.219,-99.890,170.690,39.516,157.470
C08488=1042.037,195.971,-99.865,170.687,39.515,157.470
C08489=1042.031,195.721,-99.840,170.684,39.514,157.470
C08490=1042.025,195.473,-99.817,170.682,39.512,157.469
C08491=1042.019,195.224,-99.791,170.679,39.511,157.469
C08492=1042.012,194.975,-99.767,170.676,39.510,157.469
C08493=1042.007,194.727,-99.742,170.673,39.509,157.468
C08494=1042.000,194.478,-99.718,170.671,39.508,157.468
C08495=1041.994,194.229,-99.694,170.667,39.506,157.468
C08496=1041.987,193.924,-99.663,170.664,39.505,157.467
C08497=1041.979,193.619,-99.634,170.660,39.503,157.467
C08498=1041.972,193.314,-99.604,170.657,39.502,157.466
C08499=1041.964,193.008,-99.573,170.654,39.500,157.466
C08500=1041.958,192.761,-99.549,170.651,39.499,157.466
C08501=1041.952,192.511,-99.524,170.648,39.497,157.465
C08502=1041.946,192.262,-99.500,170.646,39.496,157.465
C08503=1041.940,192.014,-99.476,170.642,39.495,157.465
C08504=1041.933,191.765,-99.451,170.640,39.493,157.464
C08505=1041.927,191.516,-99.427,170.638,39.492,157.464
C08506=1041.921,191.268,-99.403,170.634,39.491,157.464
C08507=1041.916,191.018,-99.378,170.632,39.490,157.463
C08508=1041.909,190.770,-99.355,170.629,39.489,157.463
C08509=1041.904,190.521,-99.330,170.626,39.488,157.463
C08510=1041.897,190.273,-99.305,170.624,39.486,157.462
C08511=1041.891,190.024,-99.281,170.621,39.485,157.462
C08512=1041.884,189.739,-99.254,170.617,39.483,157.461
C08513=1041.877,189.455,-99.226,170.615,39.482,157.461
C08514=1041.870,189.171,-99.199,170.612,39.481,157.461
C08515=1041.864,188.886,-99.170,170.608,39.480,157.460
C08516=1041.857,188.637,-99.146,170.606,39.478,157.460
C08517=1041.852,188.389,-99.122,170.603,39.477,157.460
C08518=1041.845,188.140,-99.098,170.600,39.476,157.459
C08519=1041.840,187.891,-99.074,170.598,39.474,157.459
C08520=1041.833,187.642,-99.050,170.595,39.473,157.459
C08521=1041.828,187.393,-99.025,170.592,39.472,157.458
C08522=1041.821,187.144,-99.001,170.590,39.471,157.458
C08523=1041.816,186.896,-98.977,170.587,39.469,157.457
C08524=1041.809,186.647,-98.953,170.584,39.468,157.457
C08525=1041.803,186.399,-98.929,170.581,39.467,157.457
C08526=1041.798,186.149,-98.905,170.579,39.465,157.456
C08527=1041.792,185.901,-98.881,170.576,39.464,157.456
C08528=1041.786,185.652,-98.856,170.573,39.463,157.456
C08529=1041.780,185.404,-98.833,170.571,39.462,157.456
C08530=1041.774,185.155,-98.808,170.568,39.461,157.455
C08531=1041.768,184.906,-98.784,170.565,39.460,157.455
C08532=1041.762,184.657,-98.760,170.563,39.458,157.455
C08533=1041.756,184.408,-98.736,170.560,39.457,157.454
C08534=1041.750,184.160,-98.712,170.557,39.456,157.454
C08535=1041.744,183.911,-98.688,170.555,39.455,157.453
C08536=1041.738,183.662,-98.664,170.552,39.454,157.453
C08537=1041.732,183.413,-98.640,170.549,39.453,157.453
C08538=1041.726,183.164,-98.617,170.547,39.451,157.453
C08539=1041.719,182.915,-98.593,170.545,39.450,157.452
C08540=1041.713,182.667,-98.569,170.541,39.449,157.452
C08541=1041.706,182.418,-98.546,170.539,39.448,157.452
C08542=1041.700,182.170,-98.523,170.536,39.447,157.451
C08543=1041.694,181.921,-98.499,170.534,39.446,157.451
C08544=1041.688,181.672,-98.476,170.531,39.445,157.451
C08545=1041.681,181.423,-98.452,170.528,39.444,157.450
C08546=1041.675,181.174,-98.428,170.526,39.443,157.450
C08547=1041.669,180.925,-98.405,170.524,39.442,157.450
C08548=1041.663,180.677,-98.381,170.520,39.441,157.450
C08549=1041.656,180.428,-98.357,170.518,39.440,157.449
C08550=1041.651,180.179,-98.334,170.515,39.439,157.449
C08551=1041.644,179.930,-98.310,170.512,39.438,157.449
C08552=1041.638,179.681,-98.286,170.510,39.437,157.448
C08553=1041.631,179.432,-98.264,170.507,39.436,157.448
C08554=1041.625,179.184,-98.240,170.505,39.435,157.448
C08555=1041.619,178.935,-98.217,170.502,39.434,157.448
C08556=1041.612,178.686,-98.193,170.499,39.433,157.447
C08557=1041.607,178.437,-98.170,170.497,39.432,157.447
C08558=1041.600,178.188,-98.146,170.494,39.431,157.447
C08559=1041.594,177.939,-98.123,170.491,39.430,157.446
C08560=1041.588,177.691,-98.099,170.489,39.429,157.446
C08561=1041.582,177.441,-98.076,170.487,39.428,157.446
C08562=1041.576,177.193,-98.052,170.483,39.427,157.446
C08563=1041.569,176.944,-98.030,170.481,39.426,157.445
C08564=1041.563,176.695,-98.006,170.479,39.425,157.445
C08565=1041.557,176.447,-97.983,170.476,39.424,157.445
C08566=1041.550,176.198,-97.959,170.473,39.423,157.444
C08567=1041.545,175.949,-97.936,170.471,39.422,157.444
C08568=1041.538,175.700,-97.912,170.469,39.421,157.444
C08569=1041.532,175.451,-97.889,170.466,39.420,157.444
C08570=1041.526,175.203,-97.865,170.463,39.419,157.443
C08571=1041.519,174.953,-97.843,170.461,39.418,157.443
C08572=1041.513,174.704,-97.820,170.458,39.417,157.443
C08573=1041.507,174.456,-97.796,170.455,39.416,157.442
C08574=1041.501,174.207,-97.773,170.453,39.415,157.442
C08575=1041.495,173.958,-97.749,170.451,39.414,157.442
C08576=1041.489,173.673,-97.723,170.448,39.413,157.442
C08577=1041.481,173.389,-97.696,170.444,39.412,157.441
C08578=1041.474,173.103,-97.669,170.442,39.411,157.441
C08579=1041.467,172.819,-97.644,170.439,39.410,157.441
C08580=1041.461,172.570,-97.620,170.436,39.409,157.440
C08581=1041.455,172.321,-97.597,170.434,39.407,157.440
C08582=1041.449,172.072,-97.574,170.431,39.406,157.440
C08583=1041.443,171.823,-97.550,170.429,39.405,157.439
C08584=1041.436,171.575,-97.527,170.426,39.404,157.439
C08585=1041.431,171.326,-97.505,170.424,39.404,157.439
C08586=1041.425,171.077,-97.481,170.421,39.403,157.439
C08587=1041.418,170.828,-97.458,170.419,39.402,157.438
C08588=1041.412,170.579,-97.435,170.416,39.401,157.438
C08589=1041.407,170.330,-97.412,170.414,39.399,157.438
C08590=1041.401,170.081,-97.389,170.411,39.398,157.437
C08591=1041.394,169.833,-97.366,170.409,39.397,157.437
C08592=1041.388,169.584,-97.342,170.406,39.397,157.437
C08593=1041.382,169.335,-97.319,170.404,39.396,157.437
C08594=1041.376,169.086,-97.296,170.401,39.395,157.436
C08595=1041.370,168.838,-97.273,170.399,39.394,157.436
C08596=1041.365,168.589,-97.250,170.396,39.393,157.436
C08597=1041.358,168.339,-97.227,170.394,39.391,157.436
C08598=1041.352,168.090,-97.204,170.392,39.390,157.435
C08599=1041.346,167.842,-97.181,170.389,39.390,157.435
C08600=1041.340,167.593,-97.158,170.386,39.389,157.435
C08601=1041.335,167.344,-97.135,170.384,39.388,157.434
C08602=1041.328,167.096,-97.112,170.382,39.387,157.434
C08603=1041.322,166.846,-97.089,170.379,39.386,157.434
C08604=1041.316,166.597,-97.066,170.376,39.385,157.434
C08605=1041.310,166.348,-97.043,170.374,39.384,157.433
C08606=1041.304,166.100,-97.020,170.372,39.383,157.433
C08607=1041.299,165.851,-96.997,170.370,39.382,157.433
C08608=1041.292,165.602,-96.975,170.367,39.381,157.433
C08609=1041.286,165.353,-96.952,170.364,39.380,157.432
C08610=1041.281,165.104,-96.929,170.362,39.379,157.432
C08611=1041.275,164.855,-96.906,170.360,39.378,157.432
C08612=1041.269,164.606,-96.883,170.357,39.377,157.431
C08613=1041.262,164.357,-96.860,170.355,39.376,157.431
C08614=1041.256,164.108,-96.837,170.353,39.375,157.431
C08615=1041.251,163.859,-96.814,170.349,39.374,157.431
C08616=1041.245,163.610,-96.791,170.347,39.373,157.430
C08617=1041.239,163.362,-96.769,170.345,39.372,157.430
C08618=1041.233,163.113,-96.746,170.343,39.371,157.430
C08619=1041.227,162.864,-96.723,170.340,39.370,157.430
C08620=1041.221,162.615,-96.700,170.338,39.369,157.429
C08621=1041.216,162.366,-96.677,170.336,39.368,157.429
C08622=1041.209,162.118,-96.655,170.333,39.367,157.429
C08623=1041.203,161.869,-96.632,170.330,39.366,157.428
C08624=1041.198,161.620,-96.609,170.328,39.365,157.428
C08625=1041.192,161.371,-96.586,170.326,39.364,157.428
C08626=1041.186,161.122,-96.563,170.324,39.363,157.428
C08627=1041.180,160.874,-96.541,170.321,39.362,157.427
C08628=1041.174,160.624,-96.519,170.319,39.361,157.427
C08629=1041.169,160.375,-96.496,170.316,39.360,157.427
C08630=1041.163,160.126,-96.473,170.314,39.359,157.427
C08631=1041.156,159.878,-96.450,170.311,39.358,157.426
C08632=1041.149,159.628,-96.428,170.309,39.358,157.426
C08633=1041.144,159.379,-96.405,170.307,39.357,157.426
C08634=1041.137,159.130,-96.383,170.305,39.356,157.425
C08635=1041.131,158.882,-96.361,170.302,39.355,157.425
C08636=1041.125,158.633,-96.338,170.299,39.354,157.425
C08637=1041.119,158.384,-96.316,170.297,39.354,157.425
C08638=1041.113,158.135,-96.293,170.295,39.353,157.425
C08639=1041.107,157.886,-96.271,170.293,39.351,157.424
C08640=1041.100,157.600,-96.246,170.289,39.351,157.424
C08641=1041.093,157.316,-96.220,170.287,39.350,157.424
C08642=1041.086,157.030,-96.195,170.284,39.349,157.423
C08643=1041.079,156.745,-96.170,170.282,39.348,157.423
C08644=1041.073,156.496,-96.147,170.279,39.347,157.423
C08645=1041.067,156.248,-96.124,170.277,39.346,157.423
C08646=1041.061,155.998,-96.102,170.274,39.345,157.422
C08647=1041.055,155.749,-96.080,170.272,39.345,157.422
C08648=1041.048,155.501,-96.057,170.269,39.344,157.422
C08649=1041.043,155.251,-96.035,170.267,39.342,157.422
C08650=1041.037,155.003,-96.013,170.265,39.342,157.422
C08651=1041.030,154.754,-95.991,170.263,39.341,157.421
C08652=1041.025,154.505,-95.968,170.261,39.340,157.421
C08653=1041.019,154.255,-95.947,170.258,39.339,157.421
C08654=1041.012,154.007,-95.924,170.255,39.339,157.421
C08655=1041.006,153.758,-95.903,170.253,39.338,157.420
C08656=1041.000,153.509,-95.880,170.251,39.337,157.420
C08657=1040.994,153.260,-95.858,170.249,39.336,157.420
C08658=1040.988,153.011,-95.836,170.246,39.335,157.420
C08659=1040.981,152.762,-95.814,170.244,39.335,157.419
C08660=1040.975,152.513,-95.792,170.242,39.334,157.419
C08661=1040.969,152.264,-95.769,170.240,39.333,157.419
C08662=1040.963,152.015,-95.747,170.236,39.332,157.419
C08663=1040.957,151.766,-95.725,170.234,39.332,157.418
C08664=1040.950,151.517,-95.703,170.232,39.330,157.418
C08665=1040.945,151.268,-95.681,170.230,39.330,157.418
C08666=1040.938,151.019,-95.658,170.228,39.329,157.418
C08667=1040.932,150.770,-95.637,170.225,39.328,157.418
C08668=1040.927,150.521,-95.616,170.223,39.327,157.417
C08669=1040.920,150.273,-95.593,170.221,39.327,157.417
C08670=1040.915,150.023,-95.571,170.219,39.326,157.417
C08671=1040.909,149.774,-95.549,170.217,39.325,157.417
C08672=1040.902,149.526,-95.527,170.213,39.324,157.416
C08673=1040.896,149.276,-95.505,170.211,39.324,157.416
C08674=1040.890,149.028,-95.483,170.209,39.323,157.416
C08675=1040.883,148.779,-95.461,170.207,39.322,157.416
C08676=1040.877,148.529,-95.440,170.204,39.321,157.415
C08677=1040.872,148.281,-95.418,170.202,39.321,157.415
C08678=1040.866,148.032,-95.396,170.200,39.319,157.415
C08679=1040.860,147.783,-95.374,170.198,39.319,157.415
C08680=1040.854,147.534,-95.352,170.196,39.318,157.415
C08681=1040.847,147.285,-95.330,170.193,39.317,157.414
C08682=1040.841,147.036,-95.308,170.191,39.316,157.414
C08683=1040.835,146.787,-95.287,170.188,39.316,157.414
C08684=1040.829,146.537,-95.265,170.186,39.315,157.414
C08685=1040.823,146.289,-95.244,170.184,39.314,157.413
C08686=1040.817,146.040,-95.221,170.182,39.314,157.413
C08687=1040.810,145.791,-95.200,170.179,39.313,157.413
C08688=1040.804,145.542,-95.178,170.177,39.312,157.413
C08689=1040.798,145.293,-95.156,170.175,39.311,157.413
C08690=1040.792,145.043,-95.135,170.173,39.311,157.412
C08691=1040.786,144.794,-95.113,170.171,39.310,157.412
C08692=1040.780,144.546,-95.091,170.168,39.309,157.412
C08693=1040.774,144.297,-95.070,170.166,39.309,157.412
C08694=1040.768,144.048,-95.048,170.164,39.307,157.411
C08695=1040.761,143.799,-95.027,170.162,39.307,157.411
C08696=1040.755,143.550,-95.005,170.159,39.307,157.411
C08697=1040.749,143.301,-94.984,170.156,39.305,157.411
C08698=1040.743,143.052,-94.962,170.154,39.305,157.411
C08699=1040.737,142.803,-94.941,170.152,39.304,157.410
C08700=1040.731,142.554,-94.919,170.150,39.303,157.410
C08701=1040.724,142.304,-94.897,170.148,39.303,157.410
C08702=1040.718,142.057,-94.875,170.145,39.302,157.410
C08703=1040.712,141.807,-94.854,170.143,39.301,157.410
C08704=1040.705,141.521,-94.829,170.141,39.300,157.409
C08705=1040.698,141.236,-94.805,170.138,39.299,157.409
C08706=1040.691,140.950,-94.780,170.135,39.299,157.409
C08707=1040.685,140.665,-94.755,170.133,39.298,157.409
C08708=1040.679,140.416,-94.734,170.131,39.297,157.408
C08709=1040.672,140.166,-94.712,170.129,39.296,157.408
C08710=1040.665,139.917,-94.691,170.127,39.295,157.408
C08711=1040.660,139.669,-94.670,170.124,39.295,157.408
C08712=1040.654,139.420,-94.648,170.122,39.294,157.407
C08713=1040.648,139.170,-94.626,170.119,39.293,157.407
C08714=1040.642,138.922,-94.605,170.117,39.293,157.407
C08715=1040.636,138.673,-94.584,170.115,39.292,157.407
C08716=1040.629,138.424,-94.562,170.113,39.291,157.407
C08717=1040.623,138.174,-94.542,170.110,39.291,157.407
C08718=1040.618,137.926,-94.520,170.108,39.290,157.406
C08719=1040.611,137.676,-94.499,170.106,39.289,157.406
C08720=1040.604,137.427,-94.478,170.104,39.289,157.406
C08721=1040.598,137.178,-94.456,170.102,39.288,157.406
C08722=1040.593,136.930,-94.435,170.099,39.287,157.405
C08723=1040.587,136.681,-94.413,170.097,39.287,157.405
C08724=1040.580,136.431,-94.393,170.095,39.286,157.405
C08725=1040.574,136.183,-94.371,170.093,39.285,157.405
C08726=1040.568,135.933,-94.350,170.091,39.285,157.405
C08727=1040.561,135.684,-94.329,170.088,39.284,157.404
C08728=1040.555,135.435,-94.307,170.086,39.283,157.404
C08729=1040.550,135.186,-94.287,170.084,39.283,157.404
C08730=1040.543,134.937,-94.266,170.082,39.281,157.404
C08731=1040.537,134.688,-94.244,170.080,39.281,157.404
C08732=1040.531,134.439,-94.223,170.078,39.280,157.403
C08733=1040.525,134.190,-94.202,170.075,39.280,157.403
C08734=1040.519,133.941,-94.181,170.073,39.279,157.403
C08735=1040.513,133.692,-94.159,170.071,39.278,157.403
C08736=1040.506,133.443,-94.138,170.069,39.278,157.403
C08737=1040.500,133.194,-94.117,170.067,39.277,157.402
C08738=1040.495,132.945,-94.096,170.064,39.276,157.402
C08739=1040.488,132.696,-94.075,170.062,39.276,157.402
C08740=1040.482,132.446,-94.054,170.060,39.275,157.402
C08741=1040.476,132.198,-94.033,170.058,39.274,157.402
C08742=1040.469,131.949,-94.012,170.056,39.274,157.401
C08743=1040.464,131.700,-93.991,170.054,39.273,157.401
C08744=1040.458,131.451,-93.970,170.051,39.272,157.401
C08745=1040.451,131.202,-93.949,170.049,39.272,157.401
C08746=1040.446,130.953,-93.928,170.047,39.271,157.401
C08747=1040.439,130.704,-93.907,170.045,39.270,157.400
C08748=1040.433,130.454,-93.886,170.043,39.270,157.400
C08749=1040.427,130.206,-93.866,170.041,39.269,157.400
C08750=1040.420,129.956,-93.845,170.038,39.269,157.400
C08751=1040.414,129.707,-93.824,170.036,39.268,157.400
C08752=1040.408,129.458,-93.804,170.034,39.268,157.400
C08753=1040.401,129.209,-93.783,170.032,39.267,157.399
C08754=1040.395,128.960,-93.761,170.030,39.266,157.399
C08755=1040.389,128.711,-93.741,170.028,39.266,157.399
C08756=1040.382,128.462,-93.721,170.025,39.265,157.399
C08757=1040.376,128.212,-93.699,170.023,39.265,157.399
C08758=1040.370,127.964,-93.679,170.021,39.264,157.398
C08759=1040.363,127.715,-93.658,170.019,39.264,157.398
C08760=1040.358,127.466,-93.637,170.017,39.262,157.398
C08761=1040.351,127.217,-93.616,170.015,39.262,157.398
C08762=1040.345,126.967,-93.596,170.012,39.261,157.398
C08763=1040.339,126.719,-93.575,170.010,39.261,157.398
C08764=1040.332,126.469,-93.554,170.008,39.261,157.397
C08765=1040.326,126.221,-93.534,170.006,39.260,157.397
C08766=1040.320,125.971,-93.513,170.004,39.259,157.397
C08767=1040.314,125.722,-93.493,170.002,39.258,157.397
C08768=1040.307,125.436,-93.469,169.998,39.258,157.397
C08769=1040.300,125.151,-93.445,169.996,39.258,157.396
C08770=1040.292,124.865,-93.421,169.994,39.256,157.396
C08771=1040.285,124.579,-93.398,169.991,39.256,157.396
C08772=1040.279,124.330,-93.377,169.989,39.256,157.396
C08773=1040.273,124.081,-93.357,169.987,39.255,157.396
C08774=1040.267,123.831,-93.336,169.984,39.254,157.395
C08775=1040.261,123.583,-93.315,169.983,39.253,157.395
C08776=1040.254,123.333,-93.295,169.981,39.253,157.395
C08777=1040.248,123.084,-93.275,169.979,39.252,157.395
C08778=1040.242,122.835,-93.253,169.977,39.252,157.395
C08779=1040.236,122.586,-93.233,169.974,39.251,157.394
C08780=1040.230,122.337,-93.213,169.972,39.250,157.394
C08781=1040.223,122.089,-93.192,169.970,39.250,157.394
C08782=1040.218,121.839,-93.171,169.968,39.249,157.394
C08783=1040.212,121.590,-93.151,169.966,39.249,157.394
C08784=1040.205,121.341,-93.131,169.964,39.248,157.394
C08785=1040.199,121.092,-93.110,169.962,39.247,157.393
C08786=1040.193,120.843,-93.089,169.959,39.247,157.393
C08787=1040.187,120.594,-93.069,169.957,39.246,157.393
C08788=1040.181,120.344,-93.049,169.955,39.246,157.393
C08789=1040.175,120.096,-93.028,169.953,39.245,157.393
C08790=1040.169,119.847,-93.008,169.951,39.244,157.392
C08791=1040.162,119.597,-92.988,169.949,39.244,157.392
C08792=1040.157,119.348,-92.967,169.946,39.243,157.392
C08793=1040.150,119.099,-92.946,169.944,39.243,157.392
C08794=1040.144,118.851,-92.926,169.942,39.242,157.392
C08795=1040.138,118.601,-92.905,169.940,39.241,157.391
C08796=1040.132,118.352,-92.885,169.938,39.241,157.391
C08797=1040.125,118.102,-92.865,169.937,39.240,157.391
C08798=1040.120,117.854,-92.845,169.934,39.240,157.391
C08799=1040.114,117.605,-92.824,169.932,39.239,157.391
C08800=1040.107,117.356,-92.803,169.930,39.238,157.391
C08801=1040.101,117.107,-92.783,169.928,39.237,157.390
C08802=1040.095,116.857,-92.762,169.926,39.237,157.390
C08803=1040.089,116.608,-92.742,169.924,39.236,157.390
C08804=1040.084,116.359,-92.722,169.921,39.236,157.390
C08805=1040.077,116.110,-92.702,169.919,39.235,157.390
C08806=1040.072,115.861,-92.682,169.917,39.234,157.389
C08807=1040.066,115.612,-92.662,169.915,39.234,157.389
C08808=1040.059,115.363,-92.641,169.913,39.233,157.389
C08809=1040.053,115.114,-92.621,169.910,39.232,157.389
C08810=1040.047,114.864,-92.600,169.909,39.232,157.389
C08811=1040.041,114.615,-92.580,169.907,39.231,157.389
C08812=1040.035,114.367,-92.560,169.905,39.231,157.388
C08813=1040.028,114.117,-92.539,169.903,39.230,157.388
C08814=1040.023,113.868,-92.519,169.901,39.229,157.388
C08815=1040.017,113.619,-92.499,169.899,39.229,157.388
C08816=1040.010,113.370,-92.479,169.896,39.228,157.388
C08817=1040.004,113.121,-92.459,169.894,39.228,157.387
C08818=1039.998,112.872,-92.439,169.892,39.227,157.387
C08819=1039.992,112.623,-92.418,169.890,39.227,157.387
C08820=1039.986,112.374,-92.398,169.888,39.226,157.387
C08821=1039.980,112.125,-92.378,169.886,39.225,157.387
C08822=1039.974,111.875,-92.359,169.883,39.225,157.387
C08823=1039.968,111.626,-92.339,169.882,39.224,157.386
C08824=1039.962,111.377,-92.319,169.880,39.223,157.386
C08825=1039.955,111.128,-92.299,169.878,39.223,157.386
C08826=1039.949,110.879,-92.279,169.876,39.222,157.386
C08827=1039.942,110.629,-92.258,169.874,39.222,157.386
C08828=1039.936,110.381,-92.238,169.872,39.222,157.386
C08829=1039.930,110.132,-92.218,169.869,39.221,157.385
C08830=1039.924,109.882,-92.199,169.867,39.221,157.385
C08831=1039.918,109.633,-92.179,169.865,39.220,157.385
C08832=1039.911,109.347,-92.157,169.863,39.220,157.385
C08833=1039.904,109.061,-92.134,169.861,39.218,157.385
C08834=1039.896,108.775,-92.111,169.858,39.218,157.385
C08835=1039.889,108.489,-92.088,169.855,39.217,157.384
C08836=1039.883,108.240,-92.068,169.853,39.217,157.384
C08837=1039.877,107.991,-92.049,169.851,39.217,157.384
C08838=1039.870,107.742,-92.028,169.849,39.216,157.384
C08839=1039.864,107.492,-92.009,169.847,39.216,157.384
C08840=1039.858,107.244,-91.989,169.845,39.215,157.384
C08841=1039.852,106.994,-91.969,169.844,39.214,157.383
C08842=1039.846,106.745,-91.949,169.841,39.214,157.383
C08843=1039.839,106.496,-91.930,169.839,39.213,157.383
C08844=1039.833,106.247,-91.910,169.837,39.213,157.383
C08845=1039.827,105.998,-91.890,169.835,39.213,157.383
C08846=1039.821,105.748,-91.871,169.833,39.212,157.383
C08847=1039.815,105.500,-91.851,169.831,39.212,157.382
C08848=1039.808,105.250,-91.831,169.828,39.210,157.382
C08849=1039.802,105.001,-91.812,169.826,39.210,157.382
C08850=1039.796,104.752,-91.792,169.824,39.209,157.382
C08851=1039.790,104.503,-91.772,169.822,39.209,157.382
C08852=1039.784,104.253,-91.752,169.820,39.208,157.382
C08853=1039.778,104.004,-91.732,169.819,39.208,157.381
C08854=1039.771,103.756,-91.713,169.817,39.207,157.381
C08855=1039.765,103.506,-91.694,169.815,39.207,157.381
C08856=1039.759,103.258,-91.674,169.812,39.206,157.381
C08857=1039.753,103.008,-91.653,169.810,39.206,157.381
C08858=1039.747,102.759,-91.634,169.808,39.205,157.381
C08859=1039.740,102.510,-91.615,169.806,39.205,157.380
C08860=1039.735,102.261,-91.595,169.804,39.204,157.380
C08861=1039.728,102.011,-91.575,169.802,39.204,157.380
C08862=1039.722,101.762,-91.556,169.800,39.203,157.380
C08863=1039.716,101.513,-91.536,169.798,39.203,157.380
C08864=1039.710,101.264,-91.517,169.796,39.202,157.379
C08865=1039.704,101.015,-91.497,169.794,39.201,157.379
C08866=1039.698,100.766,-91.477,169.792,39.201,157.379
C08867=1039.692,100.516,-91.458,169.790,39.200,157.379
C08868=1039.685,100.268,-91.438,169.788,39.200,157.379
C08869=1039.679,100.018,-91.419,169.785,39.199,157.379
C08870=1039.673,99.769,-91.399,169.783,39.199,157.379
C08871=1039.666,99.519,-91.380,169.781,39.198,157.378
C08872=1039.660,99.271,-91.360,169.779,39.198,157.378
C08873=1039.654,99.022,-91.342,169.778,39.197,157.378
C08874=1039.648,98.772,-91.322,169.776,39.197,157.378
C08875=1039.641,98.524,-91.303,169.774,39.197,157.378
C08876=1039.635,98.273,-91.283,169.772,39.196,157.378
C08877=1039.628,98.025,-91.264,169.769,39.196,157.378
C08878=1039.623,97.776,-91.245,169.767,39.195,157.377
C08879=1039.616,97.526,-91.226,169.765,39.195,157.377
C08880=1039.610,97.278,-91.206,169.763,39.194,157.377
C08881=1039.604,97.028,-91.187,169.761,39.194,157.377
C08882=1039.597,96.778,-91.168,169.759,39.193,157.377
C08883=1039.592,96.530,-91.148,169.757,39.193,157.377
C08884=1039.585,96.280,-91.129,169.754,39.192,157.376
C08885=1039.579,96.032,-91.109,169.753,39.192,157.376
C08886=1039.573,95.782,-91.091,169.751,39.191,157.376
C08887=1039.567,95.533,-91.071,169.749,39.191,157.376
C08888=1039.561,95.284,-91.053,169.747,39.190,157.376
C08889=1039.554,95.034,-91.032,169.745,39.190,157.376
C08890=1039.548,94.785,-91.014,169.743,39.189,157.376
C08891=1039.542,94.536,-90.995,169.740,39.189,157.375
C08892=1039.535,94.287,-90.975,169.738,39.188,157.375
C08893=1039.529,94.038,-90.956,169.736,39.188,157.375
C08894=1039.523,93.789,-90.937,169.735,39.187,157.375
C08895=1039.517,93.540,-90.917,169.733,39.187,157.375
C08896=1039.510,93.254,-90.896,169.730,39.186,157.375
C08897=1039.503,92.967,-90.874,169.728,39.186,157.374
C08898=1039.495,92.682,-90.852,169.725,39.185,157.374
C08899=1039.488,92.395,-90.830,169.723,39.185,157.374
C08900=1039.482,92.146,-90.810,169.721,39.184,157.374
C08901=1039.476,91.897,-90.792,169.719,39.184,157.374
C08902=1039.470,91.648,-90.772,169.717,39.183,157.374
C08903=1039.464,91.399,-90.754,169.715,39.183,157.373
C08904=1039.458,91.149,-90.734,169.714,39.182,157.373
C08905=1039.451,90.901,-90.715,169.712,39.182,157.373
C08906=1039.446,90.651,-90.696,169.709,39.181,157.373
C08907=1039.439,90.402,-90.677,169.707,39.181,157.373
C08908=1039.433,90.153,-90.658,169.705,39.180,157.373
C08909=1039.427,89.904,-90.639,169.703,39.180,157.372
C08910=1039.420,89.654,-90.620,169.701,39.179,157.372
C08911=1039.414,89.404,-90.601,169.699,39.179,157.372
C08912=1039.408,89.155,-90.582,169.697,39.178,157.372
C08913=1039.401,88.907,-90.563,169.694,39.178,157.372
C08914=1039.395,88.658,-90.544,169.693,39.177,157.372
C08915=1039.388,88.409,-90.526,169.691,39.177,157.372
C08916=1039.383,88.159,-90.506,169.689,39.177,157.372
C08917=1039.376,87.910,-90.488,169.687,39.176,157.371
C08918=1039.370,87.661,-90.469,169.685,39.176,157.371
C08919=1039.363,87.412,-90.450,169.683,39.175,157.371
C08920=1039.358,87.162,-90.431,169.681,39.175,157.371
C08921=1039.351,86.913,-90.413,169.678,39.174,157.371
C08922=1039.345,86.664,-90.394,169.676,39.174,157.371
C08923=1039.338,86.415,-90.375,169.674,39.173,157.370
C08924=1039.332,86.166,-90.357,169.672,39.174,157.370
C08925=1039.326,85.916,-90.337,169.671,39.173,157.370
C08926=1039.320,85.667,-90.319,169.669,39.173,157.370
C08927=1039.313,85.418,-90.300,169.667,39.172,157.370
C08928=1039.307,85.169,-90.281,169.665,39.172,157.370
C08929=1039.300,84.920,-90.263,169.662,39.171,157.370
C08930=1039.295,84.671,-90.244,169.660,39.171,157.369
C08931=1039.289,84.421,-90.226,169.658,39.170,157.369
C08932=1039.282,84.172,-90.207,169.656,39.170,157.369
C08933=1039.276,83.923,-90.188,169.654,39.169,157.369
C08934=1039.269,83.673,-90.170,169.653,39.169,157.369
C08935=1039.264,83.424,-90.150,169.651,39.169,157.369
C08936=1039.257,83.175,-90.132,169.649,39.168,157.369
C08937=1039.251,82.926,-90.113,169.646,39.168,157.368
C08938=1039.244,82.677,-90.094,169.644,39.167,157.368
C08939=1039.238,82.428,-90.076,169.642,39.167,157.368
C08940=1039.232,82.178,-90.057,169.640,39.166,157.368
C08941=1039.226,81.928,-90.039,169.638,39.166,157.368
C08942=1039.220,81.679,-90.020,169.636,39.165,157.368
C08943=1039.213,81.430,-90.001,169.635,39.165,157.368
C08944=1039.207,81.181,-89.983,169.632,39.164,157.367
C08945=1039.201,80.932,-89.963,169.630,39.164,157.367
C08946=1039.195,80.682,-89.945,169.628,39.163,157.367
C08947=1039.188,80.433,-89.926,169.626,39.163,157.367
C08948=1039.182,80.184,-89.908,169.624,39.163,157.367
C08949=1039.176,79.935,-89.890,169.622,39.162,157.367
C08950=1039.170,79.686,-89.871,169.620,39.162,157.367
C08951=1039.164,79.437,-89.852,169.619,39.161,157.366
C08952=1039.158,79.187,-89.833,169.616,39.161,157.366
C08953=1039.152,78.938,-89.815,169.614,39.160,157.366
C08954=1039.145,78.689,-89.797,169.612,39.160,157.366
C08955=1039.139,78.440,-89.778,169.610,39.159,157.366
C08956=1039.133,78.190,-89.760,169.608,39.159,157.366
C08957=1039.126,77.941,-89.742,169.606,39.158,157.365
C08958=1039.120,77.692,-89.723,169.604,39.158,157.365
C08959=1039.114,77.443,-89.705,169.602,39.158,157.365
C08960=1039.107,77.157,-89.683,169.599,39.157,157.365
C08961=1039.100,76.870,-89.662,169.597,39.157,157.365
C08962=1039.093,76.585,-89.641,169.595,39.156,157.365
C08963=1039.086,76.298,-89.620,169.593,39.156,157.365
C08964=1039.079,76.049,-89.602,169.591,39.155,157.364
C08965=1039.072,75.800,-89.584,169.589,39.155,157.364
C08966=1039.066,75.551,-89.565,169.587,39.154,157.364
C08967=1039.060,75.301,-89.547,169.585,39.154,157.364
C08968=1039.054,75.052,-89.529,169.582,39.153,157.364
C08969=1039.048,74.803,-89.510,169.580,39.153,157.364
C08970=1039.042,74.553,-89.492,169.578,39.153,157.364
C08971=1039.035,74.304,-89.474,169.577,39.152,157.363
C08972=1039.029,74.055,-89.456,169.575,39.152,157.363
C08973=1039.023,73.805,-89.437,169.573,39.151,157.363
C08974=1039.016,73.556,-89.419,169.571,39.151,157.363
C08975=1039.010,73.308,-89.402,169.569,39.151,157.363
C08976=1039.003,73.059,-89.383,169.567,39.151,157.363
C08977=1038.997,72.809,-89.365,169.564,39.150,157.363
C08978=1038.991,72.560,-89.346,169.562,39.150,157.362
C08979=1038.985,72.310,-89.328,169.560,39.149,157.362
C08980=1038.978,72.061,-89.310,169.559,39.148,157.362
C08981=1038.973,71.812,-89.292,169.557,39.149,157.362
C08982=1038.966,71.563,-89.274,169.555,39.148,157.362
C08983=1038.960,71.313,-89.256,169.553,39.148,157.362
C08984=1038.953,71.064,-89.238,169.551,39.147,157.362
C08985=1038.947,70.814,-89.220,169.548,39.147,157.362
C08986=1038.941,70.566,-89.201,169.546,39.146,157.361
C08987=1038.935,70.316,-89.183,169.544,39.146,157.361
C08988=1038.929,70.067,-89.165,169.542,39.146,157.361
C08989=1038.923,69.817,-89.147,169.541,39.145,157.361
C08990=1038.916,69.568,-89.129,169.539,39.145,157.361
C08991=1038.910,69.319,-89.111,169.537,39.144,157.361
C08992=1038.904,69.070,-89.093,169.535,39.144,157.361
C08993=1038.897,68.821,-89.075,169.532,39.143,157.360
C08994=1038.891,68.571,-89.057,169.530,39.143,157.360
C08995=1038.884,68.321,-89.039,169.528,39.143,157.360
C08996=1038.879,68.073,-89.021,169.526,39.142,157.360
C08997=1038.872,67.823,-89.003,169.524,39.142,157.360
C08998=1038.866,67.574,-88.985,169.522,39.141,157.360
C08999=1038.859,67.325,-88.967,169.520,39.141,157.360
C09000=1038.854,67.076,-88.950,169.519,39.141,157.360
C09001=1038.847,66.827,-88.931,169.517,39.140,157.359
C09002=1038.840,66.577,-88.914,169.514,39.140,157.359
C09003=1038.834,66.327,-88.896,169.512,39.139,157.359
C09004=1038.829,66.078,-88.878,169.510,39.139,157.359
C09005=1038.822,65.830,-88.860,169.508,39.139,157.359
C09006=1038.815,65.580,-88.842,169.506,39.138,157.359
C09007=1038.809,65.330,-88.824,169.504,39.138,157.359
C09008=1038.803,65.082,-88.806,169.502,39.138,157.359
C09009=1038.797,64.832,-88.789,169.500,39.138,157.358
C09010=1038.790,64.582,-88.771,169.499,39.137,157.358
C09011=1038.784,64.333,-88.753,169.496,39.137,157.358
C09012=1038.778,64.085,-88.735,169.494,39.136,157.358
C09013=1038.772,63.835,-88.717,169.492,39.136,157.358
C09014=1038.765,63.585,-88.700,169.490,39.136,157.358
C09015=1038.759,63.336,-88.682,169.488,39.135,157.358
C09016=1038.752,63.087,-88.665,169.486,39.135,157.358
C09017=1038.746,62.837,-88.647,169.484,39.135,157.357
C09018=1038.739,62.588,-88.629,169.482,39.134,157.357
C09019=1038.732,62.339,-88.611,169.480,39.134,157.357
C09020=1038.727,62.090,-88.594,169.478,39.134,157.357
C09021=1038.720,61.841,-88.577,169.475,39.133,157.357
C09022=1038.714,61.591,-88.559,169.473,39.134,157.357
C09023=1038.707,61.341,-88.541,169.471,39.133,157.357
C09024=1038.700,61.055,-88.521,169.469,39.133,157.357
